   LIN {X -9.322, Y 41.876, Z 87.550} C_DIS
   LIN {X -9.208, Y 43.312, Z 87.550} C_DIS
   LIN {X -9.178, Y 43.420, Z 87.550} C_DIS
   LIN {X -8.370, Y 44.918, Z 87.550} C_DIS
   LIN {X -6.846, Y 45.773, Z 87.550} C_DIS
   LIN {X -6.068, Y 46.221, Z 87.550} C_DIS
   LIN {X -5.087, Y 46.175, Z 87.550} C_DIS
   LIN {X -4.325, Y 46.141, Z 87.550}
   LaserEnd_Ext()
   LIN {X -8.280, Y 42.370, Z 87.550}
   LaserStart_Ext()
   LIN {X -8.280, Y 41.871, Z 87.550}
   LaserEnd_Ext()
   LIN {X -7.280, Y 39.330, Z 87.550}
   LaserStart_Ext()
   LIN {X -7.280, Y 44.383, Z 87.550}
   LaserEnd_Ext()
   LIN {X -6.280, Y 44.945, Z 87.550}
   LaserStart_Ext()
   LIN {X -6.280, Y 36.969, Z 87.550}
   LaserEnd_Ext()
   LIN {X -5.280, Y -20.988, Z 87.550}
   LaserStart_Ext()
   LIN {X -5.280, Y -16.273, Z 87.550}
   LaserEnd_Ext()
   LIN {X -5.280, Y 34.366, Z 87.550}
   LaserStart_Ext()
   LIN {X -5.280, Y 45.183, Z 87.550}
   LaserEnd_Ext()
   LIN {X -4.280, Y 44.988, Z 87.550}
   LaserStart_Ext()
   LIN {X -4.280, Y 31.324, Z 87.550}
   LaserEnd_Ext()
   LIN {X -4.280, Y -13.176, Z 87.550}
   LaserStart_Ext()
   LIN {X -4.280, Y -23.277, Z 87.550}
   LaserEnd_Ext()
   LIN {X -3.280, Y -24.526, Z 87.550}
   LaserStart_Ext()
   LIN {X -3.280, Y -20.919, Z 87.550}
   LaserEnd_Ext()
   LIN {X -3.280, Y -17.023, Z 87.550}
   LaserStart_Ext()
   LIN {X -3.280, Y -9.752, Z 87.550}
   LaserEnd_Ext()
   LIN {X -3.280, Y 27.844, Z 87.550}
   LaserStart_Ext()
   LIN {X -3.280, Y 44.352, Z 87.550}
   LaserEnd_Ext()
   LIN {X -2.280, Y 42.864, Z 87.550}
   LaserStart_Ext()
   LIN {X -2.280, Y 23.421, Z 87.550}
   LaserEnd_Ext()
   LIN {X -2.280, Y -5.420, Z 87.550}
   LaserStart_Ext()
   LIN {X -2.280, Y -15.048, Z 87.550}
   LaserEnd_Ext()
   LIN {X -2.280, Y -22.581, Z 87.550}
   LaserStart_Ext()
   LIN {X -2.280, Y -25.295, Z 87.550}
   LaserEnd_Ext()
   LIN {X -1.280, Y -25.911, Z 87.550}
   LaserStart_Ext()
   LIN {X -1.280, Y -23.637, Z 87.550}
   LaserEnd_Ext()
   LIN {X -1.280, Y -13.980, Z 87.550}
   LaserStart_Ext()
   LIN {X -1.280, Y 1.203, Z 87.550}
   LaserEnd_Ext()
   LIN {X -1.280, Y 16.034, Z 87.550}
   LaserStart_Ext()
   LIN {X -1.280, Y 40.953, Z 87.550}
   LaserEnd_Ext()
   LIN {X -0.280, Y 38.939, Z 87.550}
   LaserStart_Ext()
   LIN {X -0.280, Y -13.537, Z 87.550}
   LaserEnd_Ext()
   LIN {X -0.280, Y -24.134, Z 87.550}
   LaserStart_Ext()
   LIN {X -0.280, Y -26.154, Z 87.550}
   LaserEnd_Ext()
   LIN {X 0.720, Y -26.397, Z 87.550}
   LaserStart_Ext()
   LIN {X 0.720, Y -24.611, Z 87.550}
   LaserEnd_Ext()
   LIN {X 0.720, Y -13.095, Z 87.550}
   LaserStart_Ext()
   LIN {X 0.720, Y 36.811, Z 87.550}
   LaserEnd_Ext()
   LIN {X 1.720, Y 34.552, Z 87.550}
   LaserStart_Ext()
   LIN {X 1.720, Y -12.865, Z 87.550}
   LaserEnd_Ext()
   LIN {X 1.720, Y -24.679, Z 87.550}
   LaserStart_Ext()
   LIN {X 1.720, Y -26.645, Z 87.550}
   LaserEnd_Ext()
   LIN {X 2.720, Y -26.731, Z 87.550}
   LaserStart_Ext()
   LIN {X 2.720, Y -24.716, Z 87.550}
   LaserEnd_Ext()
   LIN {X 2.720, Y -12.903, Z 87.550}
   LaserStart_Ext()
   LIN {X 2.720, Y 32.147, Z 87.550}
   LaserEnd_Ext()
   LIN {X 3.720, Y 29.606, Z 87.550}
   LaserStart_Ext()
   LIN {X 3.720, Y -12.955, Z 87.550}
   LaserEnd_Ext()
   LIN {X 3.720, Y -24.543, Z 87.550}
   LaserStart_Ext()
   LIN {X 3.720, Y -26.549, Z 87.550}
   LaserEnd_Ext()
   LIN {X 4.720, Y -26.367, Z 87.550}
   LaserStart_Ext()
   LIN {X 4.720, Y -24.134, Z 87.550}
   LaserEnd_Ext()
   LIN {X 4.720, Y -13.416, Z 87.550}
   LaserStart_Ext()
   LIN {X 4.720, Y 26.609, Z 87.550}
   LaserEnd_Ext()
   LIN {X 5.720, Y 23.635, Z 87.550}
   LaserStart_Ext()
   LIN {X 5.720, Y -13.918, Z 87.550}
   LaserEnd_Ext()
   LIN {X 5.720, Y -23.685, Z 87.550}
   LaserStart_Ext()
   LIN {X 5.720, Y -25.868, Z 87.550}
   LaserEnd_Ext()
   LIN {X 6.720, Y -25.325, Z 87.550}
   LaserStart_Ext()
   LIN {X 6.720, Y -22.621, Z 87.550}
   LaserEnd_Ext()
   LIN {X 6.720, Y -14.966, Z 87.550}
   LaserStart_Ext()
   LIN {X 6.720, Y 20.268, Z 87.550}
   LaserEnd_Ext()
   LIN {X 7.720, Y 16.143, Z 87.550}
   LaserStart_Ext()
   LIN {X 7.720, Y -16.327, Z 87.550}
   LaserEnd_Ext()
   LIN {X 7.720, Y -21.000, Z 87.550}
   LaserStart_Ext()
   LIN {X 7.720, Y -24.463, Z 87.550}
   LaserEnd_Ext()
   LIN {X 8.720, Y -23.296, Z 87.550}
   LaserStart_Ext()
   LIN {X 8.720, Y 12.020, Z 87.550}
   LaserEnd_Ext()
   LIN {X 9.720, Y 5.409, Z 87.550}
   LaserStart_Ext()
   LIN {X 9.720, Y -21.071, Z 87.550}
   LaserEnd_Ext()
   LIN {X 10.720, Y -10.941, Z 87.550}
   LaserStart_Ext()
   LIN {X 10.720, Y -7.263, Z 87.550}
   LaserEnd_Ext()
   LIN {X -2.101, Y -21.081, Z 88.400}
   LaserStart_Ext()
   LIN {X -2.327, Y -20.250, Z 88.400} C_DIS
   LIN {X -2.653, Y -19.069, Z 88.400} C_DIS
   LIN {X -2.140, Y -16.745, Z 88.400} C_DIS
   LIN {X -2.058, Y -16.383, Z 88.400} C_DIS
   LIN {X -1.960, Y -16.269, Z 88.400} C_DIS
   LIN {X -0.730, Y -14.804, Z 88.400} C_DIS
   LIN {X 1.550, Y -13.800, Z 88.400} C_DIS
   LIN {X 2.406, Y -13.830, Z 88.400} C_DIS
   LIN {X 3.592, Y -13.874, Z 88.400} C_DIS
   LIN {X 4.404, Y -14.282, Z 88.400} C_DIS
   LIN {X 5.494, Y -14.823, Z 88.400} C_DIS
   LIN {X 6.466, Y -16.137, Z 88.400} C_DIS
   LIN {X 7.004, Y -16.869, Z 88.400} C_DIS
   LIN {X 7.127, Y -17.688, Z 88.400} C_DIS
   LIN {X 7.338, Y -19.054, Z 88.400} C_DIS
   LIN {X 6.967, Y -20.266, Z 88.400} C_DIS
   LIN {X 6.671, Y -21.222, Z 88.400} C_DIS
   LIN {X 5.735, Y -22.242, Z 88.400} C_DIS
   LIN {X 5.196, Y -22.834, Z 88.400} C_DIS
   LIN {X 4.756, Y -23.018, Z 88.400} C_DIS
   LIN {X 3.171, Y -23.668, Z 88.400} C_DIS
   LIN {X 1.356, Y -23.607, Z 88.400} C_DIS
   LIN {X 1.086, Y -23.596, Z 88.400} C_DIS
   LIN {X 0.744, Y -23.427, Z 88.400} C_DIS
   LIN {X -0.767, Y -22.681, Z 88.400} C_DIS
   LIN {X -1.591, Y -21.695, Z 88.400} C_DIS
   LIN {X -2.101, Y -21.081, Z 88.400}
   LaserEnd_Ext()
   LIN {X -1.865, Y -26.739, Z 88.400}
   LaserStart_Ext()
   LIN {X -2.207, Y -26.496, Z 88.400} C_DIS
   LIN {X -4.280, Y -24.904, Z 88.400} C_DIS
   LIN {X -5.389, Y -23.237, Z 88.400} C_DIS
   LIN {X -5.889, Y -22.475, Z 88.400} C_DIS
   LIN {X -6.157, Y -21.214, Z 88.400} C_DIS
   LIN {X -6.672, Y -18.848, Z 88.400} C_DIS
   LIN {X -6.289, Y -16.613, Z 88.400} C_DIS
   LIN {X -6.132, Y -15.724, Z 88.400} C_DIS
   LIN {X -5.888, Y -15.002, Z 88.400} C_DIS
   LIN {X -5.036, Y -12.454, Z 88.400} C_DIS
   LIN {X -4.260, Y -9.716, Z 88.400} C_DIS
   LIN {X -4.130, Y -9.256, Z 88.400} C_DIS
   LIN {X -4.052, Y -8.927, Z 88.400} C_DIS
   LIN {X -3.419, Y -6.256, Z 88.400} C_DIS
   LIN {X -3.129, Y -4.745, Z 88.400} C_DIS
   LIN {X -2.837, Y -3.225, Z 88.400} C_DIS
   LIN {X -2.519, Y -1.124, Z 88.400} C_DIS
   LIN {X -2.431, Y -0.548, Z 88.400} C_DIS
   LIN {X -1.994, Y 3.966, Z 88.400} C_DIS
   LIN {X -1.892, Y 5.625, Z 88.400} C_DIS
   LIN {X -1.905, Y 12.231, Z 88.400} C_DIS
   LIN {X -2.343, Y 17.044, Z 88.400} C_DIS
   LIN {X -3.185, Y 22.879, Z 88.400} C_DIS
   LIN {X -4.399, Y 28.248, Z 88.400} C_DIS
   LIN {X -4.637, Y 29.079, Z 88.400} C_DIS
   LIN {X -5.862, Y 32.955, Z 88.400} C_DIS
   LIN {X -5.956, Y 33.234, Z 88.400} C_DIS
   LIN {X -6.386, Y 34.380, Z 88.400} C_DIS
   LIN {X -6.924, Y 35.827, Z 88.400} C_DIS
   LIN {X -7.316, Y 36.776, Z 88.400} C_DIS
   LIN {X -7.831, Y 38.016, Z 88.400} C_DIS
   LIN {X -8.303, Y 39.073, Z 88.400} C_DIS
   LIN {X -8.483, Y 39.477, Z 88.400} C_DIS
   LIN {X -8.577, Y 39.682, Z 88.400} C_DIS
   LIN {X -9.008, Y 40.612, Z 88.400} C_DIS
   LIN {X -9.347, Y 41.838, Z 88.400} C_DIS
   LIN {X -9.397, Y 42.016, Z 88.400} C_DIS
   LIN {X -9.375, Y 42.239, Z 88.400} C_DIS
   LIN {X -9.262, Y 43.429, Z 88.400} C_DIS
   LIN {X -8.453, Y 44.892, Z 88.400} C_DIS
   LIN {X -8.396, Y 44.998, Z 88.400} C_DIS
   LIN {X -8.295, Y 45.059, Z 88.400} C_DIS
   LIN {X -6.140, Y 46.258, Z 88.400} C_DIS
   LIN {X -5.430, Y 46.228, Z 88.400} C_DIS
   LIN {X -4.398, Y 46.181, Z 88.400} C_DIS
   LIN {X -3.166, Y 45.535, Z 88.400} C_DIS
   LIN {X -2.858, Y 45.374, Z 88.400} C_DIS
   LIN {X -2.697, Y 45.180, Z 88.400} C_DIS
   LIN {X -1.925, Y 44.237, Z 88.400} C_DIS
   LIN {X -1.257, Y 43.001, Z 88.400} C_DIS
   LIN {X -1.154, Y 42.804, Z 88.400} C_DIS
   LIN {X -0.334, Y 41.232, Z 88.400} C_DIS
   LIN {X 0.389, Y 39.778, Z 88.400} C_DIS
   LIN {X 0.732, Y 39.087, Z 88.400} C_DIS
   LIN {X 0.977, Y 38.576, Z 88.400} C_DIS
   LIN {X 2.267, Y 35.768, Z 88.400} C_DIS
   LIN {X 2.837, Y 34.460, Z 88.400} C_DIS
   LIN {X 4.233, Y 31.014, Z 88.400} C_DIS
   LIN {X 4.570, Y 30.191, Z 88.400} C_DIS
   LIN {X 4.734, Y 29.722, Z 88.400} C_DIS
   LIN {X 7.364, Y 21.900, Z 88.400} C_DIS
   LIN {X 8.161, Y 18.532, Z 88.400} C_DIS
   LIN {X 9.659, Y 12.653, Z 88.400} C_DIS
   LIN {X 10.596, Y 6.682, Z 88.400} C_DIS
   LIN {X 11.255, Y 1.954, Z 88.400} C_DIS
   LIN {X 11.382, Y -0.482, Z 88.400} C_DIS
   LIN {X 11.492, Y -1.843, Z 88.400} C_DIS
   LIN {X 11.725, Y -4.721, Z 88.400} C_DIS
   LIN {X 11.784, Y -8.079, Z 88.400} C_DIS
   LIN {X 11.812, Y -9.507, Z 88.400} C_DIS
   LIN {X 11.807, Y -9.910, Z 88.400} C_DIS
   LIN {X 11.734, Y -13.310, Z 88.400} C_DIS
   LIN {X 11.644, Y -15.135, Z 88.400} C_DIS
   LIN {X 11.582, Y -16.267, Z 88.400} C_DIS
   LIN {X 11.486, Y -17.425, Z 88.400} C_DIS
   LIN {X 11.326, Y -19.519, Z 88.400} C_DIS
   LIN {X 10.716, Y -21.461, Z 88.400} C_DIS
   LIN {X 10.154, Y -23.186, Z 88.400} C_DIS
   LIN {X 8.060, Y -25.630, Z 88.400} C_DIS
   LIN {X 7.954, Y -25.756, Z 88.400} C_DIS
   LIN {X 7.764, Y -25.857, Z 88.400} C_DIS
   LIN {X 5.067, Y -27.308, Z 88.400} C_DIS
   LIN {X 3.728, Y -27.551, Z 88.400} C_DIS
   LIN {X 1.570, Y -27.601, Z 88.400} C_DIS
   LIN {X -1.865, Y -26.739, Z 88.400}
   LaserEnd_Ext()
   LIN {X 4.690, Y -26.360, Z 88.400}
   LaserStart_Ext()
   LIN {X 0.734, Y -26.360, Z 88.400}
   LaserEnd_Ext()
   LIN {X -2.044, Y -25.360, Z 88.400}
   LaserStart_Ext()
   LIN {X 6.576, Y -25.360, Z 88.400}
   LaserEnd_Ext()
   LIN {X 7.832, Y -24.360, Z 88.400}
   LaserStart_Ext()
   LIN {X 4.118, Y -24.360, Z 88.400}
   LaserEnd_Ext()
   LIN {X 0.375, Y -24.360, Z 88.400}
   LaserStart_Ext()
   LIN {X -3.346, Y -24.360, Z 88.400}
   LaserEnd_Ext()
   LIN {X -4.106, Y -23.360, Z 88.400}
   LaserStart_Ext()
   LIN {X -1.499, Y -23.360, Z 88.400}
   LaserEnd_Ext()
   LIN {X 6.070, Y -23.360, Z 88.400}
   LaserStart_Ext()
   LIN {X 8.688, Y -23.360, Z 88.400}
   LaserEnd_Ext()
   LIN {X 9.371, Y -22.360, Z 88.400}
   LaserStart_Ext()
   LIN {X 6.984, Y -22.360, Z 88.400}
   LaserEnd_Ext()
   LIN {X -2.339, Y -22.360, Z 88.400}
   LaserStart_Ext()
   LIN {X -4.768, Y -22.360, Z 88.400}
   LaserEnd_Ext()
   LIN {X -5.103, Y -21.360, Z 88.400}
   LaserStart_Ext()
   LIN {X -3.060, Y -21.360, Z 88.400}
   LaserEnd_Ext()
   LIN {X 7.675, Y -21.360, Z 88.400}
   LaserStart_Ext()
   LIN {X 9.697, Y -21.360, Z 88.400}
   LaserEnd_Ext()
   LIN {X 10.014, Y -20.360, Z 88.400}
   LaserStart_Ext()
   LIN {X 7.984, Y -20.360, Z 88.400}
   LaserEnd_Ext()
   LIN {X -3.334, Y -20.360, Z 88.400}
   LaserStart_Ext()
   LIN {X -5.319, Y -20.360, Z 88.400}
   LaserEnd_Ext()
   LIN {X -5.537, Y -19.360, Z 88.400}
   LaserStart_Ext()
   LIN {X -3.610, Y -19.360, Z 88.400}
   LaserEnd_Ext()
   LIN {X 8.290, Y -19.360, Z 88.400}
   LaserStart_Ext()
   LIN {X 10.328, Y -19.360, Z 88.400}
   LaserEnd_Ext()
   LIN {X 10.412, Y -18.360, Z 88.400}
   LaserStart_Ext()
   LIN {X 8.243, Y -18.360, Z 88.400}
   LaserEnd_Ext()
   LIN {X -3.521, Y -18.360, Z 88.400}
   LaserStart_Ext()
   LIN {X -5.574, Y -18.360, Z 88.400}
   LaserEnd_Ext()
   LIN {X -5.402, Y -17.360, Z 88.400}
   LaserStart_Ext()
   LIN {X -3.300, Y -17.360, Z 88.400}
   LaserEnd_Ext()
   LIN {X 8.089, Y -17.360, Z 88.400}
   LaserStart_Ext()
   LIN {X 10.488, Y -17.360, Z 88.400}
   LaserEnd_Ext()
   LIN {X 10.571, Y -16.360, Z 88.400}
   LaserStart_Ext()
   LIN {X 7.864, Y -16.360, Z 88.400}
   LaserEnd_Ext()
   LIN {X -3.078, Y -16.360, Z 88.400}
   LaserStart_Ext()
   LIN {X -5.228, Y -16.360, Z 88.400}
   LaserEnd_Ext()
   LIN {X -4.953, Y -15.360, Z 88.400}
   LaserStart_Ext()
   LIN {X -2.503, Y -15.360, Z 88.400}
   LaserEnd_Ext()
   LIN {X 7.135, Y -15.360, Z 88.400}
   LaserStart_Ext()
   LIN {X 10.630, Y -15.360, Z 88.400}
   LaserEnd_Ext()
   LIN {X 10.681, Y -14.360, Z 88.400}
   LaserStart_Ext()
   LIN {X 6.395, Y -14.360, Z 88.400}
   LaserEnd_Ext()
   LIN {X -1.663, Y -14.360, Z 88.400}
   LaserStart_Ext()
   LIN {X -4.619, Y -14.360, Z 88.400}
   LaserEnd_Ext()
   LIN {X -4.284, Y -13.360, Z 88.400}
   LaserStart_Ext()
   LIN {X 0.068, Y -13.360, Z 88.400}
   LaserEnd_Ext()
   LIN {X 4.797, Y -13.360, Z 88.400}
   LaserStart_Ext()
   LIN {X 10.730, Y -13.360, Z 88.400}
   LaserEnd_Ext()
   LIN {X 10.754, Y -12.360, Z 88.400}
   LaserStart_Ext()
   LIN {X -3.970, Y -12.360, Z 88.400}
   LaserEnd_Ext()
   LIN {X -3.687, Y -11.360, Z 88.400}
   LaserStart_Ext()
   LIN {X 10.775, Y -11.360, Z 88.400}
   LaserEnd_Ext()
   LIN {X 10.797, Y -10.360, Z 88.400}
   LaserStart_Ext()
   LIN {X -3.403, Y -10.360, Z 88.400}
   LaserEnd_Ext()
   LIN {X -3.127, Y -9.360, Z 88.400}
   LaserStart_Ext()
   LIN {X 10.809, Y -9.360, Z 88.400}
   LaserEnd_Ext()
   LIN {X 10.789, Y -8.360, Z 88.400}
   LaserStart_Ext()
   LIN {X -2.890, Y -8.360, Z 88.400}
   LaserEnd_Ext()
   LIN {X -2.653, Y -7.360, Z 88.400}
   LaserStart_Ext()
   LIN {X 10.771, Y -7.360, Z 88.400}
   LaserEnd_Ext()
   LIN {X 10.754, Y -6.360, Z 88.400}
   LaserStart_Ext()
   LIN {X -2.421, Y -6.360, Z 88.400}
   LaserEnd_Ext()
   LIN {X -2.229, Y -5.360, Z 88.400}
   LaserStart_Ext()
   LIN {X 10.736, Y -5.360, Z 88.400}
   LaserEnd_Ext()
   LIN {X 10.693, Y -4.360, Z 88.400}
   LaserStart_Ext()
   LIN {X -2.037, Y -4.360, Z 88.400}
   LaserEnd_Ext()
   LIN {X -1.846, Y -3.360, Z 88.400}
   LaserStart_Ext()
   LIN {X 10.612, Y -3.360, Z 88.400}
   LaserEnd_Ext()
   LIN {X 10.531, Y -2.360, Z 88.400}
   LaserStart_Ext()
   LIN {X -1.694, Y -2.360, Z 88.400}
   LaserEnd_Ext()
   LIN {X -1.543, Y -1.360, Z 88.400}
   LaserStart_Ext()
   LIN {X 10.450, Y -1.360, Z 88.400}
   LaserEnd_Ext()
   LIN {X 10.375, Y -0.360, Z 88.400}
   LaserStart_Ext()
   LIN {X -1.408, Y -0.360, Z 88.400}
   LaserEnd_Ext()
   LIN {X -1.311, Y 0.640, Z 88.400}
   LaserStart_Ext()
   LIN {X 10.322, Y 0.640, Z 88.400}
   LaserEnd_Ext()
   LIN {X 10.270, Y 1.640, Z 88.400}
   LaserStart_Ext()
   LIN {X -1.214, Y 1.640, Z 88.400}
   LaserEnd_Ext()
   LIN {X -1.118, Y 2.640, Z 88.400}
   LaserStart_Ext()
   LIN {X 10.149, Y 2.640, Z 88.400}
   LaserEnd_Ext()
   LIN {X 10.010, Y 3.640, Z 88.400}
   LaserStart_Ext()
   LIN {X -1.021, Y 3.640, Z 88.400}
   LaserEnd_Ext()
   LIN {X -0.951, Y 4.640, Z 88.400}
   LaserStart_Ext()
   LIN {X 9.871, Y 4.640, Z 88.400}
   LaserEnd_Ext()
   LIN {X 9.732, Y 5.640, Z 88.400}
   LaserStart_Ext()
   LIN {X -0.892, Y 5.640, Z 88.400}
   LaserEnd_Ext()
   LIN {X -0.894, Y 6.640, Z 88.400}
   LaserStart_Ext()
   LIN {X 9.591, Y 6.640, Z 88.400}
   LaserEnd_Ext()
   LIN {X 9.434, Y 7.640, Z 88.400}
   LaserStart_Ext()
   LIN {X -0.896, Y 7.640, Z 88.400}
   LaserEnd_Ext()
   LIN {X -0.898, Y 8.640, Z 88.400}
   LaserStart_Ext()
   LIN {X 9.277, Y 8.640, Z 88.400}
   LaserEnd_Ext()
   LIN {X 9.120, Y 9.640, Z 88.400}
   LaserStart_Ext()
   LIN {X -0.900, Y 9.640, Z 88.400}
   LaserEnd_Ext()
   LIN {X -0.902, Y 10.640, Z 88.400}
   LaserStart_Ext()
   LIN {X 8.963, Y 10.640, Z 88.400}
   LaserEnd_Ext()
   LIN {X 8.806, Y 11.640, Z 88.400}
   LaserStart_Ext()
   LIN {X -0.904, Y 11.640, Z 88.400}
   LaserEnd_Ext()
   LIN {X -0.938, Y 12.640, Z 88.400}
   LaserStart_Ext()
   LIN {X 8.630, Y 12.640, Z 88.400}
   LaserEnd_Ext()
   LIN {X 8.376, Y 13.640, Z 88.400}
   LaserStart_Ext()
   LIN {X -1.029, Y 13.640, Z 88.400}
   LaserEnd_Ext()
   LIN {X -1.120, Y 14.640, Z 88.400}
   LaserStart_Ext()
   LIN {X 8.121, Y 14.640, Z 88.400}
   LaserEnd_Ext()
   LIN {X 7.866, Y 15.640, Z 88.400}
   LaserStart_Ext()
   LIN {X -1.211, Y 15.640, Z 88.400}
   LaserEnd_Ext()
   LIN {X -1.302, Y 16.640, Z 88.400}
   LaserStart_Ext()
   LIN {X 7.611, Y 16.640, Z 88.400}
   LaserEnd_Ext()
   LIN {X 7.356, Y 17.640, Z 88.400}
   LaserStart_Ext()
   LIN {X -1.419, Y 17.640, Z 88.400}
   LaserEnd_Ext()
   LIN {X -1.563, Y 18.640, Z 88.400}
   LaserStart_Ext()
   LIN {X 7.108, Y 18.640, Z 88.400}
   LaserEnd_Ext()
   LIN {X 6.871, Y 19.640, Z 88.400}
   LaserStart_Ext()
   LIN {X -1.707, Y 19.640, Z 88.400}
   LaserEnd_Ext()
   LIN {X -1.852, Y 20.640, Z 88.400}
   LaserStart_Ext()
   LIN {X 6.635, Y 20.640, Z 88.400}
   LaserEnd_Ext()
   LIN {X 6.397, Y 21.640, Z 88.400}
   LaserStart_Ext()
   LIN {X -1.996, Y 21.640, Z 88.400}
   LaserEnd_Ext()
   LIN {X -2.141, Y 22.640, Z 88.400}
   LaserStart_Ext()
   LIN {X 6.060, Y 22.640, Z 88.400}
   LaserEnd_Ext()
   LIN {X 5.724, Y 23.640, Z 88.400}
   LaserStart_Ext()
   LIN {X -2.332, Y 23.640, Z 88.400}
   LaserEnd_Ext()
   LIN {X -2.558, Y 24.640, Z 88.400}
   LaserStart_Ext()
   LIN {X 5.388, Y 24.640, Z 88.400}
   LaserEnd_Ext()
   LIN {X 5.052, Y 25.640, Z 88.400}
   LaserStart_Ext()
   LIN {X -2.784, Y 25.640, Z 88.400}
   LaserEnd_Ext()
   LIN {X -3.010, Y 26.640, Z 88.400}
   LaserStart_Ext()
   LIN {X 4.715, Y 26.640, Z 88.400}
   LaserEnd_Ext()
   LIN {X 4.379, Y 27.640, Z 88.400}
   LaserStart_Ext()
   LIN {X -3.237, Y 27.640, Z 88.400}
   LaserEnd_Ext()
   LIN {X -3.471, Y 28.640, Z 88.400}
   LaserStart_Ext()
   LIN {X 4.043, Y 28.640, Z 88.400}
   LaserEnd_Ext()
   LIN {X 3.703, Y 29.640, Z 88.400}
   LaserStart_Ext()
   LIN {X -3.766, Y 29.640, Z 88.400}
   LaserEnd_Ext()
   LIN {X -4.082, Y 30.640, Z 88.400}
   LaserStart_Ext()
   LIN {X 3.306, Y 30.640, Z 88.400}
   LaserEnd_Ext()
   LIN {X 2.900, Y 31.640, Z 88.400}
   LaserStart_Ext()
   LIN {X -4.398, Y 31.640, Z 88.400}
   LaserEnd_Ext()
   LIN {X -4.714, Y 32.640, Z 88.400}
   LaserStart_Ext()
   LIN {X 2.495, Y 32.640, Z 88.400}
   LaserEnd_Ext()
   LIN {X 2.090, Y 33.640, Z 88.400}
   LaserStart_Ext()
   LIN {X -5.040, Y 33.640, Z 88.400}
   LaserEnd_Ext()
   LIN {X -5.415, Y 34.640, Z 88.400}
   LaserStart_Ext()
   LIN {X 1.668, Y 34.640, Z 88.400}
   LaserEnd_Ext()
   LIN {X 1.226, Y 35.640, Z 88.400}
   LaserStart_Ext()
   LIN {X -5.788, Y 35.640, Z 88.400}
   LaserEnd_Ext()
   LIN {X -6.178, Y 36.640, Z 88.400}
   LaserStart_Ext()
   LIN {X 0.766, Y 36.640, Z 88.400}
   LaserEnd_Ext()
   LIN {X 0.306, Y 37.640, Z 88.400}
   LaserStart_Ext()
   LIN {X -6.592, Y 37.640, Z 88.400}
   LaserEnd_Ext()
   LIN {X -7.014, Y 38.640, Z 88.400}
   LaserStart_Ext()
   LIN {X -0.163, Y 38.640, Z 88.400}
   LaserEnd_Ext()
   LIN {X -0.659, Y 39.640, Z 88.400}
   LaserStart_Ext()
   LIN {X -7.461, Y 39.640, Z 88.400}
   LaserEnd_Ext()
   LIN {X -7.919, Y 40.640, Z 88.400}
   LaserStart_Ext()
   LIN {X -1.156, Y 40.640, Z 88.400}
   LaserEnd_Ext()
   LIN {X -1.674, Y 41.640, Z 88.400}
   LaserStart_Ext()
   LIN {X -8.255, Y 41.640, Z 88.400}
   LaserEnd_Ext()
   LIN {X -8.333, Y 42.640, Z 88.400}
   LaserStart_Ext()
   LIN {X -2.199, Y 42.640, Z 88.400}
   LaserEnd_Ext()
   LIN {X -2.739, Y 43.640, Z 88.400}
   LaserStart_Ext()
   LIN {X -8.003, Y 43.640, Z 88.400}
   LaserEnd_Ext()
   LIN {X -6.992, Y 44.640, Z 88.400}
   LaserStart_Ext()
   LIN {X -3.612, Y 44.640, Z 88.400}
   LaserEnd_Ext()
   LIN {X -1.592, Y -21.537, Z 89.250}
   LaserStart_Ext()
   LIN {X -2.015, Y -21.035, Z 89.250} C_DIS
   LIN {X -2.194, Y -20.394, Z 89.250} C_DIS
   LIN {X -2.572, Y -19.024, Z 89.250} C_DIS
   LIN {X -2.278, Y -17.692, Z 89.250} C_DIS
   LIN {X -1.967, Y -16.308, Z 89.250} C_DIS
   LIN {X -0.892, Y -15.038, Z 89.250} C_DIS
   LIN {X -0.644, Y -14.743, Z 89.250} C_DIS
   LIN {X 1.620, Y -13.745, Z 89.250} C_DIS
   LIN {X 3.253, Y -13.802, Z 89.250} C_DIS
   LIN {X 3.661, Y -13.815, Z 89.250} C_DIS
   LIN {X 4.151, Y -14.057, Z 89.250} C_DIS
   LIN {X 5.565, Y -14.759, Z 89.250} C_DIS
   LIN {X 6.551, Y -16.091, Z 89.250} C_DIS
   LIN {X 7.080, Y -16.801, Z 89.250} C_DIS
   LIN {X 7.186, Y -17.471, Z 89.250} C_DIS
   LIN {X 7.420, Y -18.985, Z 89.250} C_DIS
   LIN {X 6.909, Y -20.653, Z 89.250} C_DIS
   LIN {X 6.757, Y -21.155, Z 89.250} C_DIS
   LIN {X 6.481, Y -21.460, Z 89.250} C_DIS
   LIN {X 5.289, Y -22.769, Z 89.250} C_DIS
   LIN {X 3.705, Y -23.429, Z 89.250} C_DIS
   LIN {X 3.268, Y -23.608, Z 89.250} C_DIS
   LIN {X 2.586, Y -23.585, Z 89.250} C_DIS
   LIN {X 1.178, Y -23.542, Z 89.250} C_DIS
   LIN {X 0.300, Y -23.114, Z 89.250} C_DIS
   LIN {X -0.677, Y -22.631, Z 89.250} C_DIS
   LIN {X -1.592, Y -21.537, Z 89.250}
   LaserEnd_Ext()
   LIN {X -5.998, Y 33.271, Z 89.250}
   LaserStart_Ext()
   LIN {X -5.632, Y 32.183, Z 89.250} C_DIS
   LIN {X -4.767, Y 29.446, Z 89.250} C_DIS
   LIN {X -4.321, Y 27.887, Z 89.250} C_DIS
   LIN {X -3.278, Y 23.278, Z 89.250} C_DIS
   LIN {X -2.195, Y 15.771, Z 89.250} C_DIS
   LIN {X -1.905, Y 12.581, Z 89.250} C_DIS
   LIN {X -1.889, Y 5.163, Z 89.250} C_DIS
   LIN {X -1.949, Y 4.193, Z 89.250} C_DIS
   LIN {X -2.359, Y -0.048, Z 89.250} C_DIS
   LIN {X -2.418, Y -0.675, Z 89.250} C_DIS
   LIN {X -2.505, Y -1.257, Z 89.250} C_DIS
   LIN {X -2.823, Y -3.356, Z 89.250} C_DIS
   LIN {X -2.949, Y -4.013, Z 89.250} C_DIS
   LIN {X -3.404, Y -6.387, Z 89.250} C_DIS
   LIN {X -3.835, Y -8.202, Z 89.250} C_DIS
   LIN {X -4.113, Y -9.379, Z 89.250} C_DIS
   LIN {X -4.579, Y -11.021, Z 89.250} C_DIS
   LIN {X -5.020, Y -12.577, Z 89.250} C_DIS
   LIN {X -5.817, Y -14.962, Z 89.250} C_DIS
   LIN {X -6.058, Y -15.688, Z 89.250} C_DIS
   LIN {X -6.170, Y -16.361, Z 89.250} C_DIS
   LIN {X -6.591, Y -18.813, Z 89.250} C_DIS
   LIN {X -5.908, Y -21.949, Z 89.250} C_DIS
   LIN {X -5.799, Y -22.438, Z 89.250} C_DIS
   LIN {X -5.547, Y -22.814, Z 89.250} C_DIS
   LIN {X -4.184, Y -24.863, Z 89.250} C_DIS
   LIN {X -2.991, Y -25.779, Z 89.250} C_DIS
   LIN {X -1.597, Y -26.769, Z 89.250} C_DIS
   LIN {X 1.038, Y -27.430, Z 89.250} C_DIS
   LIN {X 4.803, Y -27.343, Z 89.250} C_DIS
   LIN {X 4.970, Y -27.313, Z 89.250} C_DIS
   LIN {X 5.307, Y -27.132, Z 89.250} C_DIS
   LIN {X 7.191, Y -26.181, Z 89.250} C_DIS
   LIN {X 8.065, Y -25.674, Z 89.250} C_DIS
   LIN {X 9.619, Y -23.837, Z 89.250} C_DIS
   LIN {X 10.254, Y -23.096, Z 89.250} C_DIS
   LIN {X 10.425, Y -22.572, Z 89.250} C_DIS
   LIN {X 11.409, Y -19.441, Z 89.250} C_DIS
   LIN {X 11.649, Y -16.305, Z 89.250} C_DIS
   LIN {X 11.657, Y -16.188, Z 89.250} C_DIS
   LIN {X 11.665, Y -16.024, Z 89.250} C_DIS
   LIN {X 11.802, Y -13.231, Z 89.250} C_DIS
   LIN {X 11.847, Y -11.119, Z 89.250} C_DIS
   LIN {X 11.872, Y -9.427, Z 89.250} C_DIS
   LIN {X 11.785, Y -5.074, Z 89.250} C_DIS
   LIN {X 11.773, Y -4.642, Z 89.250} C_DIS
   LIN {X 11.733, Y -4.149, Z 89.250} C_DIS
   LIN {X 11.468, Y -0.870, Z 89.250} C_DIS
   LIN {X 11.383, Y 0.176, Z 89.250} C_DIS
   LIN {X 11.285, Y 2.048, Z 89.250} C_DIS
   LIN {X 10.779, Y 5.683, Z 89.250} C_DIS
   LIN {X 9.699, Y 12.567, Z 89.250} C_DIS
   LIN {X 7.971, Y 19.344, Z 89.250} C_DIS
   LIN {X 7.360, Y 21.930, Z 89.250} C_DIS
   LIN {X 5.341, Y 27.934, Z 89.250} C_DIS
   LIN {X 4.513, Y 30.308, Z 89.250} C_DIS
   LIN {X 2.805, Y 34.476, Z 89.250} C_DIS
   LIN {X 2.660, Y 34.835, Z 89.250} C_DIS
   LIN {X 2.600, Y 34.972, Z 89.250} C_DIS
   LIN {X 2.284, Y 35.660, Z 89.250} C_DIS
   LIN {X 0.845, Y 38.792, Z 89.250} C_DIS
   LIN {X 0.072, Y 40.342, Z 89.250} C_DIS
   LIN {X -0.395, Y 41.282, Z 89.250} C_DIS
   LIN {X -0.599, Y 41.673, Z 89.250} C_DIS
   LIN {X -1.285, Y 42.979, Z 89.250} C_DIS
   LIN {X -1.937, Y 44.181, Z 89.250} C_DIS
   LIN {X -1.992, Y 44.283, Z 89.250} C_DIS
   LIN {X -2.078, Y 44.387, Z 89.250} C_DIS
   LIN {X -2.928, Y 45.418, Z 89.250} C_DIS
   LIN {X -4.144, Y 46.053, Z 89.250} C_DIS
   LIN {X -4.470, Y 46.221, Z 89.250} C_DIS
   LIN {X -5.183, Y 46.251, Z 89.250} C_DIS
   LIN {X -6.213, Y 46.294, Z 89.250} C_DIS
   LIN {X -6.786, Y 45.975, Z 89.250} C_DIS
   LIN {X -8.564, Y 44.907, Z 89.250} C_DIS
   LIN {X -9.211, Y 43.703, Z 89.250} C_DIS
   LIN {X -9.330, Y 43.445, Z 89.250} C_DIS
   LIN {X -9.352, Y 43.152, Z 89.250} C_DIS
   LIN {X -9.459, Y 42.045, Z 89.250} C_DIS
   LIN {X -9.087, Y 40.713, Z 89.250} C_DIS
   LIN {X -9.048, Y 40.601, Z 89.250} C_DIS
   LIN {X -8.539, Y 39.508, Z 89.250} C_DIS
   LIN {X -8.096, Y 38.522, Z 89.250} C_DIS
   LIN {X -7.884, Y 38.049, Z 89.250} C_DIS
   LIN {X -7.522, Y 37.175, Z 89.250} C_DIS
   LIN {X -6.972, Y 35.861, Z 89.250} C_DIS
   LIN {X -6.433, Y 34.432, Z 89.250} C_DIS
   LIN {X -5.998, Y 33.271, Z 89.250}
   LaserEnd_Ext()
   LIN {X 10.602, Y -2.568, Z 89.250}
   LaserStart_Ext()
   LIN {X 10.602, Y -16.881, Z 89.250}
   LaserEnd_Ext()
   LIN {X 9.602, Y -21.855, Z 89.250}
   LaserStart_Ext()
   LIN {X 9.602, Y 6.733, Z 89.250}
   LaserEnd_Ext()
   LIN {X 8.602, Y 12.821, Z 89.250}
   LaserStart_Ext()
   LIN {X 8.602, Y -23.491, Z 89.250}
   LaserEnd_Ext()
   LIN {X 7.602, Y -24.674, Z 89.250}
   LaserStart_Ext()
   LIN {X 7.602, Y -21.687, Z 89.250}
   LaserEnd_Ext()
   LIN {X 7.602, Y -15.828, Z 89.250}
   LaserStart_Ext()
   LIN {X 7.602, Y 16.744, Z 89.250}
   LaserEnd_Ext()
   LIN {X 6.602, Y 20.790, Z 89.250}
   LaserStart_Ext()
   LIN {X 6.602, Y -14.479, Z 89.250}
   LaserEnd_Ext()
   LIN {X 6.602, Y -22.812, Z 89.250}
   LaserStart_Ext()
   LIN {X 6.602, Y -25.358, Z 89.250}
   LaserEnd_Ext()
   LIN {X 5.602, Y -25.863, Z 89.250}
   LaserStart_Ext()
   LIN {X 5.602, Y -23.722, Z 89.250}
   LaserEnd_Ext()
   LIN {X 5.602, Y -13.661, Z 89.250}
   LaserStart_Ext()
   LIN {X 5.602, Y 24.020, Z 89.250}
   LaserEnd_Ext()
   LIN {X 4.602, Y 26.993, Z 89.250}
   LaserStart_Ext()
   LIN {X 4.602, Y -13.164, Z 89.250}
   LaserEnd_Ext()
   LIN {X 4.602, Y -24.138, Z 89.250}
   LaserStart_Ext()
   LIN {X 4.602, Y -26.348, Z 89.250}
   LaserEnd_Ext()
   LIN {X 3.602, Y -26.371, Z 89.250}
   LaserStart_Ext()
   LIN {X 3.602, Y -24.549, Z 89.250}
   LaserEnd_Ext()
   LIN {X 3.602, Y -12.812, Z 89.250}
   LaserStart_Ext()
   LIN {X 3.602, Y 29.884, Z 89.250}
   LaserEnd_Ext()
   LIN {X 2.602, Y 32.335, Z 89.250}
   LaserStart_Ext()
   LIN {X 2.602, Y -12.779, Z 89.250}
   LaserEnd_Ext()
   LIN {X 2.602, Y -24.586, Z 89.250}
   LaserStart_Ext()
   LIN {X 2.602, Y -26.394, Z 89.250}
   LaserEnd_Ext()
   LIN {X 1.602, Y -26.417, Z 89.250}
   LaserStart_Ext()
   LIN {X 1.602, Y -24.556, Z 89.250}
   LaserEnd_Ext()
   LIN {X 1.602, Y -12.746, Z 89.250}
   LaserStart_Ext()
   LIN {X 1.602, Y 34.749, Z 89.250}
   LaserEnd_Ext()
   LIN {X 0.602, Y 36.926, Z 89.250}
   LaserStart_Ext()
   LIN {X 0.602, Y -13.101, Z 89.250}
   LaserEnd_Ext()
   LIN {X 0.602, Y -24.374, Z 89.250}
   LaserStart_Ext()
   LIN {X 0.602, Y -26.289, Z 89.250}
   LaserEnd_Ext()
   LIN {X -0.398, Y -26.039, Z 89.250}
   LaserStart_Ext()
   LIN {X -0.398, Y -23.884, Z 89.250}
   LaserEnd_Ext()
   LIN {X -0.398, Y -13.542, Z 89.250}
   LaserStart_Ext()
   LIN {X -0.398, Y 39.045, Z 89.250}
   LaserEnd_Ext()
   LIN {X -1.398, Y 41.044, Z 89.250}
   LaserStart_Ext()
   LIN {X -1.398, Y 17.252, Z 89.250}
   LaserEnd_Ext()
   LIN {X -1.398, Y -0.512, Z 89.250}
   LaserStart_Ext()
   LIN {X -1.398, Y -14.087, Z 89.250}
   LaserEnd_Ext()
   LIN {X -1.398, Y -23.323, Z 89.250}
   LaserStart_Ext()
   LIN {X -1.398, Y -25.684, Z 89.250}
   LaserEnd_Ext()
   LIN {X -2.398, Y -24.974, Z 89.250}
   LaserStart_Ext()
   LIN {X -2.398, Y -22.133, Z 89.250}
   LaserEnd_Ext()
   LIN {X -2.398, Y -15.270, Z 89.250}
   LaserStart_Ext()
   LIN {X -2.398, Y -6.448, Z 89.250}
   LaserEnd_Ext()
   LIN {X -2.398, Y 23.919, Z 89.250}
   LaserStart_Ext()
   LIN {X -2.398, Y 42.934, Z 89.250}
   LaserEnd_Ext()
   LIN {X -3.398, Y 44.416, Z 89.250}
   LaserStart_Ext()
   LIN {X -3.398, Y 28.299, Z 89.250}
   LaserEnd_Ext()
   LIN {X -3.398, Y -10.523, Z 89.250}
   LaserStart_Ext()
   LIN {X -3.398, Y -18.128, Z 89.250}
   LaserEnd_Ext()
   LIN {X -3.398, Y -19.788, Z 89.250}
   LaserStart_Ext()
   LIN {X -3.398, Y -24.206, Z 89.250}
   LaserEnd_Ext()
   LIN {X -4.398, Y -22.736, Z 89.250}
   LaserStart_Ext()
   LIN {X -4.398, Y -13.871, Z 89.250}
   LaserEnd_Ext()
   LIN {X -4.398, Y 31.598, Z 89.250}
   LaserStart_Ext()
   LIN {X -4.398, Y 45.057, Z 89.250}
   LaserEnd_Ext()
   LIN {X -5.398, Y 45.259, Z 89.250}
   LaserStart_Ext()
   LIN {X -5.398, Y 34.519, Z 89.250}
   LaserEnd_Ext()
   LIN {X -5.398, Y -17.776, Z 89.250}
   LaserStart_Ext()
   LIN {X -5.398, Y -19.590, Z 89.250}
   LaserEnd_Ext()
   LIN {X -6.398, Y 37.080, Z 89.250}
   LaserStart_Ext()
   LIN {X -6.398, Y 45.042, Z 89.250}
   LaserEnd_Ext()
   LIN {X -7.398, Y 44.441, Z 89.250}
   LaserStart_Ext()
   LIN {X -7.398, Y 39.409, Z 89.250}
   LaserEnd_Ext()
   LIN {X -8.398, Y 41.962, Z 89.250}
   LaserStart_Ext()
   LIN {X -8.398, Y 42.631, Z 89.250}
   LaserEnd_Ext()
   LIN {X -0.588, Y -22.582, Z 90.100}
   LaserStart_Ext()
   LIN {X -0.706, Y -22.442, Z 90.100} C_DIS
   LIN {X -1.929, Y -20.988, Z 90.100} C_DIS
   LIN {X -2.435, Y -19.175, Z 90.100} C_DIS
   LIN {X -2.490, Y -18.979, Z 90.100} C_DIS
   LIN {X -2.411, Y -18.632, Z 90.100} C_DIS
   LIN {X -1.870, Y -16.222, Z 90.100} C_DIS
   LIN {X -1.137, Y -15.356, Z 90.100} C_DIS
   LIN {X -0.541, Y -14.668, Z 90.100} C_DIS
   LIN {X 1.101, Y -13.949, Z 90.100} C_DIS
   LIN {X 1.689, Y -13.690, Z 90.100} C_DIS
   LIN {X 2.048, Y -13.702, Z 90.100} C_DIS
   LIN {X 3.731, Y -13.755, Z 90.100} C_DIS
   LIN {X 5.545, Y -14.650, Z 90.100} C_DIS
   LIN {X 5.637, Y -14.695, Z 90.100} C_DIS
   LIN {X 5.712, Y -14.795, Z 90.100} C_DIS
   LIN {X 7.157, Y -16.733, Z 90.100} C_DIS
   LIN {X 7.477, Y -18.758, Z 90.100} C_DIS
   LIN {X 7.501, Y -18.916, Z 90.100} C_DIS
   LIN {X 7.448, Y -19.090, Z 90.100} C_DIS
   LIN {X 6.839, Y -21.095, Z 90.100} C_DIS
   LIN {X 5.739, Y -22.311, Z 90.100} C_DIS
   LIN {X 5.381, Y -22.704, Z 90.100} C_DIS
   LIN {X 4.557, Y -23.047, Z 90.100} C_DIS
   LIN {X 3.363, Y -23.549, Z 90.100} C_DIS
   LIN {X 2.587, Y -23.528, Z 90.100} C_DIS
   LIN {X 1.270, Y -23.488, Z 90.100} C_DIS
   LIN {X -0.388, Y -22.678, Z 90.100} C_DIS
   LIN {X -0.588, Y -22.582, Z 90.100}
   LaserEnd_Ext()
   LIN {X 5.947, Y 26.147, Z 90.100}
   LaserStart_Ext()
   LIN {X 4.456, Y 30.426, Z 90.100} C_DIS
   LIN {X 2.760, Y 34.563, Z 90.100} C_DIS
   LIN {X 2.404, Y 35.337, Z 90.100} C_DIS
   LIN {X 2.319, Y 35.520, Z 90.100} C_DIS
   LIN {X 2.137, Y 35.913, Z 90.100} C_DIS
   LIN {X 0.791, Y 38.845, Z 90.100} C_DIS
   LIN {X 0.241, Y 39.946, Z 90.100} C_DIS
   LIN {X -0.455, Y 41.332, Z 90.100} C_DIS
   LIN {X -1.225, Y 42.790, Z 90.100} C_DIS
   LIN {X -1.349, Y 43.027, Z 90.100} C_DIS
   LIN {X -1.417, Y 43.152, Z 90.100} C_DIS
   LIN {X -2.059, Y 44.329, Z 90.100} C_DIS
   LIN {X -2.945, Y 45.398, Z 90.100} C_DIS
   LIN {X -3.137, Y 45.533, Z 90.100} C_DIS
   LIN {X -4.542, Y 46.261, Z 90.100} C_DIS
   LIN {X -5.406, Y 46.297, Z 90.100} C_DIS
   LIN {X -6.285, Y 46.330, Z 90.100} C_DIS
   LIN {X -8.269, Y 45.094, Z 90.100} C_DIS
   LIN {X -8.733, Y 44.816, Z 90.100} C_DIS
   LIN {X -8.819, Y 44.655, Z 90.100} C_DIS
   LIN {X -9.432, Y 43.321, Z 90.100} C_DIS
   LIN {X -9.512, Y 42.273, Z 90.100} C_DIS
   LIN {X -9.519, Y 42.051, Z 90.100} C_DIS
   LIN {X -9.451, Y 41.825, Z 90.100} C_DIS
   LIN {X -9.126, Y 40.671, Z 90.100} C_DIS
   LIN {X -8.666, Y 39.690, Z 90.100} C_DIS
   LIN {X -8.596, Y 39.538, Z 90.100} C_DIS
   LIN {X -8.461, Y 39.239, Z 90.100} C_DIS
   LIN {X -7.937, Y 38.081, Z 90.100} C_DIS
   LIN {X -7.273, Y 36.500, Z 90.100} C_DIS
   LIN {X -7.020, Y 35.895, Z 90.100} C_DIS
   LIN {X -6.721, Y 35.101, Z 90.100} C_DIS
   LIN {X -6.041, Y 33.311, Z 90.100} C_DIS
   LIN {X -5.401, Y 31.410, Z 90.100} C_DIS
   LIN {X -4.896, Y 29.812, Z 90.100} C_DIS
   LIN {X -4.242, Y 27.527, Z 90.100} C_DIS
   LIN {X -3.371, Y 23.677, Z 90.100} C_DIS
   LIN {X -2.046, Y 14.497, Z 90.100} C_DIS
   LIN {X -1.904, Y 12.930, Z 90.100} C_DIS
   LIN {X -1.886, Y 4.701, Z 90.100} C_DIS
   LIN {X -1.904, Y 4.420, Z 90.100} C_DIS
   LIN {X -2.022, Y 3.193, Z 90.100} C_DIS
   LIN {X -2.377, Y -0.611, Z 90.100} C_DIS
   LIN {X -2.406, Y -0.844, Z 90.100} C_DIS
   LIN {X -2.783, Y -3.326, Z 90.100} C_DIS
   LIN {X -2.808, Y -3.487, Z 90.100} C_DIS
   LIN {X -2.910, Y -4.018, Z 90.100} C_DIS
   LIN {X -3.390, Y -6.517, Z 90.100} C_DIS
   LIN {X -3.617, Y -7.478, Z 90.100} C_DIS
   LIN {X -4.096, Y -9.502, Z 90.100} C_DIS
   LIN {X -4.898, Y -12.326, Z 90.100} C_DIS
   LIN {X -5.004, Y -12.700, Z 90.100} C_DIS
   LIN {X -5.195, Y -13.272, Z 90.100} C_DIS
   LIN {X -5.984, Y -15.651, Z 90.100} C_DIS
   LIN {X -6.352, Y -17.858, Z 90.100} C_DIS
   LIN {X -6.509, Y -18.778, Z 90.100} C_DIS
   LIN {X -6.253, Y -19.953, Z 90.100} C_DIS
   LIN {X -5.709, Y -22.400, Z 90.100} C_DIS
   LIN {X -4.447, Y -24.283, Z 90.100} C_DIS
   LIN {X -4.089, Y -24.821, Z 90.100} C_DIS
   LIN {X -3.775, Y -25.062, Z 90.100} C_DIS
   LIN {X -1.328, Y -26.799, Z 90.100} C_DIS
   LIN {X 0.505, Y -27.259, Z 90.100} C_DIS
   LIN {X 3.411, Y -27.192, Z 90.100} C_DIS
   LIN {X 5.286, Y -27.177, Z 90.100} C_DIS
   LIN {X 6.489, Y -26.570, Z 90.100} C_DIS
   LIN {X 8.177, Y -25.593, Z 90.100} C_DIS
   LIN {X 10.035, Y -23.396, Z 90.100} C_DIS
   LIN {X 10.398, Y -22.916, Z 90.100} C_DIS
   LIN {X 10.645, Y -22.057, Z 90.100} C_DIS
   LIN {X 11.492, Y -19.362, Z 90.100} C_DIS
   LIN {X 11.639, Y -17.436, Z 90.100} C_DIS
   LIN {X 11.733, Y -16.109, Z 90.100} C_DIS
   LIN {X 11.817, Y -14.242, Z 90.100} C_DIS
   LIN {X 11.871, Y -13.152, Z 90.100} C_DIS
   LIN {X 11.888, Y -12.328, Z 90.100} C_DIS
   LIN {X 11.931, Y -9.348, Z 90.100} C_DIS
   LIN {X 11.877, Y -6.642, Z 90.100} C_DIS
   LIN {X 11.821, Y -4.563, Z 90.100} C_DIS
   LIN {X 11.629, Y -2.190, Z 90.100} C_DIS
   LIN {X 11.443, Y 0.103, Z 90.100} C_DIS
   LIN {X 11.384, Y 0.834, Z 90.100} C_DIS
   LIN {X 11.316, Y 2.143, Z 90.100} C_DIS
   LIN {X 10.962, Y 4.684, Z 90.100} C_DIS
   LIN {X 9.738, Y 12.481, Z 90.100} C_DIS
   LIN {X 7.782, Y 20.157, Z 90.100} C_DIS
   LIN {X 7.356, Y 21.960, Z 90.100} C_DIS
   LIN {X 5.947, Y 26.147, Z 90.100}
   LaserEnd_Ext()
   LIN {X -3.518, Y 44.522, Z 90.100}
   LaserStart_Ext()
   LIN {X -7.297, Y 44.522, Z 90.100}
   LaserEnd_Ext()
   LIN {X -8.239, Y 43.522, Z 90.100}
   LaserStart_Ext()
   LIN {X -2.758, Y 43.522, Z 90.100}
   LaserEnd_Ext()
   LIN {X -2.214, Y 42.522, Z 90.100}
   LaserStart_Ext()
   LIN {X -8.490, Y 42.522, Z 90.100}
   LaserEnd_Ext()
   LIN {X -8.327, Y 41.522, Z 90.100}
   LaserStart_Ext()
   LIN {X -1.686, Y 41.522, Z 90.100}
   LaserEnd_Ext()
   LIN {X -1.167, Y 40.522, Z 90.100}
   LaserStart_Ext()
   LIN {X -7.952, Y 40.522, Z 90.100}
   LaserEnd_Ext()
   LIN {X -7.491, Y 39.522, Z 90.100}
   LaserStart_Ext()
   LIN {X -0.665, Y 39.522, Z 90.100}
   LaserEnd_Ext()
   LIN {X -0.166, Y 38.522, Z 90.100}
   LaserStart_Ext()
   LIN {X -7.039, Y 38.522, Z 90.100}
   LaserEnd_Ext()
   LIN {X -6.618, Y 37.522, Z 90.100}
   LaserStart_Ext()
   LIN {X 0.298, Y 37.522, Z 90.100}
   LaserEnd_Ext()
   LIN {X 0.757, Y 36.522, Z 90.100}
   LaserStart_Ext()
   LIN {X -6.198, Y 36.522, Z 90.100}
   LaserEnd_Ext()
   LIN {X -5.811, Y 35.522, Z 90.100}
   LaserStart_Ext()
   LIN {X 1.216, Y 35.522, Z 90.100}
   LaserEnd_Ext()
   LIN {X 1.678, Y 34.522, Z 90.100}
   LaserStart_Ext()
   LIN {X -5.431, Y 34.522, Z 90.100}
   LaserEnd_Ext()
   LIN {X -5.057, Y 33.522, Z 90.100}
   LaserStart_Ext()
   LIN {X 2.106, Y 33.522, Z 90.100}
   LaserEnd_Ext()
   LIN {X 2.516, Y 32.522, Z 90.100}
   LaserStart_Ext()
   LIN {X -4.720, Y 32.522, Z 90.100}
   LaserEnd_Ext()
   LIN {X -4.388, Y 31.522, Z 90.100}
   LaserStart_Ext()
   LIN {X 2.926, Y 31.522, Z 90.100}
   LaserEnd_Ext()
   LIN {X 3.336, Y 30.522, Z 90.100}
   LaserStart_Ext()
   LIN {X -4.072, Y 30.522, Z 90.100}
   LaserEnd_Ext()
   LIN {X -3.773, Y 29.522, Z 90.100}
   LaserStart_Ext()
   LIN {X 3.712, Y 29.522, Z 90.100}
   LaserEnd_Ext()
   LIN {X 4.060, Y 28.522, Z 90.100}
   LaserStart_Ext()
   LIN {X -3.486, Y 28.522, Z 90.100}
   LaserEnd_Ext()
   LIN {X -3.215, Y 27.522, Z 90.100}
   LaserStart_Ext()
   LIN {X 4.409, Y 27.522, Z 90.100}
   LaserEnd_Ext()
   LIN {X 4.758, Y 26.522, Z 90.100}
   LaserStart_Ext()
   LIN {X -2.989, Y 26.522, Z 90.100}
   LaserEnd_Ext()
   LIN {X -2.763, Y 25.522, Z 90.100}
   LaserStart_Ext()
   LIN {X 5.102, Y 25.522, Z 90.100}
   LaserEnd_Ext()
   LIN {X 5.439, Y 24.522, Z 90.100}
   LaserStart_Ext()
   LIN {X -2.537, Y 24.522, Z 90.100}
   LaserEnd_Ext()
   LIN {X -2.339, Y 23.522, Z 90.100}
   LaserStart_Ext()
   LIN {X 5.775, Y 23.522, Z 90.100}
   LaserEnd_Ext()
   LIN {X 6.111, Y 22.522, Z 90.100}
   LaserStart_Ext()
   LIN {X -2.194, Y 22.522, Z 90.100}
   LaserEnd_Ext()
   LIN {X -2.050, Y 21.522, Z 90.100}
   LaserStart_Ext()
   LIN {X 6.431, Y 21.522, Z 90.100}
   LaserEnd_Ext()
   LIN {X 6.668, Y 20.522, Z 90.100}
   LaserStart_Ext()
   LIN {X -1.905, Y 20.522, Z 90.100}
   LaserEnd_Ext()
   LIN {X -1.761, Y 19.522, Z 90.100}
   LaserStart_Ext()
   LIN {X 6.912, Y 19.522, Z 90.100}
   LaserEnd_Ext()
   LIN {X 7.167, Y 18.522, Z 90.100}
   LaserStart_Ext()
   LIN {X -1.617, Y 18.522, Z 90.100}
   LaserEnd_Ext()
   LIN {X -1.472, Y 17.522, Z 90.100}
   LaserStart_Ext()
   LIN {X 7.421, Y 17.522, Z 90.100}
   LaserEnd_Ext()
   LIN {X 7.676, Y 16.522, Z 90.100}
   LaserStart_Ext()
   LIN {X -1.328, Y 16.522, Z 90.100}
   LaserEnd_Ext()
   LIN {X -1.184, Y 15.522, Z 90.100}
   LaserStart_Ext()
   LIN {X 7.931, Y 15.522, Z 90.100}
   LaserEnd_Ext()
   LIN {X 8.186, Y 14.522, Z 90.100}
   LaserStart_Ext()
   LIN {X -1.044, Y 14.522, Z 90.100}
   LaserEnd_Ext()
   LIN {X -0.953, Y 13.522, Z 90.100}
   LaserStart_Ext()
   LIN {X 8.441, Y 13.522, Z 90.100}
   LaserEnd_Ext()
   LIN {X 8.696, Y 12.522, Z 90.100}
   LaserStart_Ext()
   LIN {X -0.903, Y 12.522, Z 90.100}
   LaserEnd_Ext()
   LIN {X -0.901, Y 11.522, Z 90.100}
   LaserStart_Ext()
   LIN {X 8.876, Y 11.522, Z 90.100}
   LaserEnd_Ext()
   LIN {X 9.033, Y 10.522, Z 90.100}
   LaserStart_Ext()
   LIN {X -0.899, Y 10.522, Z 90.100}
   LaserEnd_Ext()
   LIN {X -0.896, Y 9.522, Z 90.100}
   LaserStart_Ext()
   LIN {X 9.190, Y 9.522, Z 90.100}
   LaserEnd_Ext()
   LIN {X 9.347, Y 8.522, Z 90.100}
   LaserStart_Ext()
   LIN {X -0.894, Y 8.522, Z 90.100}
   LaserEnd_Ext()
   LIN {X -0.892, Y 7.522, Z 90.100}
   LaserStart_Ext()
   LIN {X 9.504, Y 7.522, Z 90.100}
   LaserEnd_Ext()
   LIN {X 9.661, Y 6.522, Z 90.100}
   LaserStart_Ext()
   LIN {X -0.890, Y 6.522, Z 90.100}
   LaserEnd_Ext()
   LIN {X -0.888, Y 5.522, Z 90.100}
   LaserStart_Ext()
   LIN {X 9.818, Y 5.522, Z 90.100}
   LaserEnd_Ext()
   LIN {X 9.975, Y 4.522, Z 90.100}
   LaserStart_Ext()
   LIN {X -0.895, Y 4.522, Z 90.100}
   LaserEnd_Ext()
   LIN {X -0.986, Y 3.522, Z 90.100}
   LaserStart_Ext()
   LIN {X 10.114, Y 3.522, Z 90.100}
   LaserEnd_Ext()
   LIN {X 10.253, Y 2.522, Z 90.100}
   LaserStart_Ext()
   LIN {X -1.081, Y 2.522, Z 90.100}
   LaserEnd_Ext()
   LIN {X -1.174, Y 1.522, Z 90.100}
   LaserStart_Ext()
   LIN {X 10.347, Y 1.522, Z 90.100}
   LaserEnd_Ext()
   LIN {X 10.406, Y 0.522, Z 90.100}
   LaserStart_Ext()
   LIN {X -1.267, Y 0.522, Z 90.100}
   LaserEnd_Ext()
   LIN {X -1.360, Y -0.478, Z 90.100}
   LaserStart_Ext()
   LIN {X 10.487, Y -0.478, Z 90.100}
   LaserEnd_Ext()
   LIN {X 10.568, Y -1.478, Z 90.100}
   LaserStart_Ext()
   LIN {X -1.491, Y -1.478, Z 90.100}
   LaserEnd_Ext()
   LIN {X -1.643, Y -2.478, Z 90.100}
   LaserStart_Ext()
   LIN {X 10.649, Y -2.478, Z 90.100}
   LaserEnd_Ext()
   LIN {X 10.730, Y -3.478, Z 90.100}
   LaserStart_Ext()
   LIN {X -1.795, Y -3.478, Z 90.100}
   LaserEnd_Ext()
   LIN {X -1.980, Y -4.478, Z 90.100}
   LaserStart_Ext()
   LIN {X 10.811, Y -4.478, Z 90.100}
   LaserEnd_Ext()
   LIN {X 10.845, Y -5.478, Z 90.100}
   LaserStart_Ext()
   LIN {X -2.172, Y -5.478, Z 90.100}
   LaserEnd_Ext()
   LIN {X -2.364, Y -6.478, Z 90.100}
   LaserStart_Ext()
   LIN {X 10.872, Y -6.478, Z 90.100}
   LaserEnd_Ext()
   LIN {X 10.894, Y -7.478, Z 90.100}
   LaserStart_Ext()
   LIN {X -2.590, Y -7.478, Z 90.100}
   LaserEnd_Ext()
   LIN {X -2.826, Y -8.478, Z 90.100}
   LaserStart_Ext()
   LIN {X 10.914, Y -8.478, Z 90.100}
   LaserEnd_Ext()
   LIN {X 10.929, Y -9.478, Z 90.100}
   LaserStart_Ext()
   LIN {X -3.063, Y -9.478, Z 90.100}
   LaserEnd_Ext()
   LIN {X -3.333, Y -10.478, Z 90.100}
   LaserStart_Ext()
   LIN {X 10.915, Y -10.478, Z 90.100}
   LaserEnd_Ext()
   LIN {X 10.900, Y -11.478, Z 90.100}
   LaserStart_Ext()
   LIN {X -3.618, Y -11.478, Z 90.100}
   LaserEnd_Ext()
   LIN {X -3.902, Y -12.478, Z 90.100}
   LaserStart_Ext()
   LIN {X 10.885, Y -12.478, Z 90.100}
   LaserEnd_Ext()
   LIN {X 10.853, Y -13.478, Z 90.100}
   LaserStart_Ext()
   LIN {X 5.430, Y -13.478, Z 90.100}
   LaserEnd_Ext()
   LIN {X -0.317, Y -13.478, Z 90.100}
   LaserStart_Ext()
   LIN {X -4.210, Y -13.478, Z 90.100}
   LaserEnd_Ext()
   LIN {X -4.542, Y -14.478, Z 90.100}
   LaserStart_Ext()
   LIN {X -1.699, Y -14.478, Z 90.100}
   LaserEnd_Ext()
   LIN {X 6.723, Y -14.478, Z 90.100}
   LaserStart_Ext()
   LIN {X 10.805, Y -14.478, Z 90.100}
   LaserEnd_Ext()
   LIN {X 10.760, Y -15.478, Z 90.100}
   LaserStart_Ext()
   LIN {X 7.469, Y -15.478, Z 90.100}
   LaserEnd_Ext()
   LIN {X -2.551, Y -15.478, Z 90.100}
   LaserStart_Ext()
   LIN {X -4.873, Y -15.478, Z 90.100}
   LaserEnd_Ext()
   LIN {X -5.108, Y -16.478, Z 90.100}
   LaserStart_Ext()
   LIN {X -2.952, Y -16.478, Z 90.100}
   LaserEnd_Ext()
   LIN {X 8.123, Y -16.478, Z 90.100}
   LaserStart_Ext()
   LIN {X 10.704, Y -16.478, Z 90.100}
   LaserEnd_Ext()
   LIN {X 10.633, Y -17.478, Z 90.100}
   LaserStart_Ext()
   LIN {X 8.287, Y -17.478, Z 90.100}
   LaserEnd_Ext()
   LIN {X -3.177, Y -17.478, Z 90.100}
   LaserStart_Ext()
   LIN {X -5.275, Y -17.478, Z 90.100}
   LaserEnd_Ext()
   LIN {X -5.443, Y -18.478, Z 90.100}
   LaserStart_Ext()
   LIN {X -3.402, Y -18.478, Z 90.100}
   LaserEnd_Ext()
   LIN {X 8.445, Y -18.478, Z 90.100}
   LaserStart_Ext()
   LIN {X 10.557, Y -18.478, Z 90.100}
   LaserEnd_Ext()
   LIN {X 10.407, Y -19.478, Z 90.100}
   LaserStart_Ext()
   LIN {X 8.375, Y -19.478, Z 90.100}
   LaserEnd_Ext()
   LIN {X -3.388, Y -19.478, Z 90.100}
   LaserStart_Ext()
   LIN {X -5.333, Y -19.478, Z 90.100}
   LaserEnd_Ext()
   LIN {X -5.112, Y -20.478, Z 90.100}
   LaserStart_Ext()
   LIN {X -3.109, Y -20.478, Z 90.100}
   LaserEnd_Ext()
   LIN {X 8.072, Y -20.478, Z 90.100}
   LaserStart_Ext()
   LIN {X 10.093, Y -20.478, Z 90.100}
   LaserEnd_Ext()
   LIN {X 9.779, Y -21.478, Z 90.100}
   LaserStart_Ext()
   LIN {X 7.763, Y -21.478, Z 90.100}
   LaserEnd_Ext()
   LIN {X -2.799, Y -21.478, Z 90.100}
   LaserStart_Ext()
   LIN {X -4.890, Y -21.478, Z 90.100}
   LaserEnd_Ext()
   LIN {X -4.453, Y -22.478, Z 90.100}
   LaserStart_Ext()
   LIN {X -1.982, Y -22.478, Z 90.100}
   LaserEnd_Ext()
   LIN {X 6.936, Y -22.478, Z 90.100}
   LaserStart_Ext()
   LIN {X 9.475, Y -22.478, Z 90.100}
   LaserEnd_Ext()
   LIN {X 8.655, Y -23.478, Z 90.100}
   LaserStart_Ext()
   LIN {X 6.011, Y -23.478, Z 90.100}
   LaserEnd_Ext()
   LIN {X -1.030, Y -23.478, Z 90.100}
   LaserStart_Ext()
   LIN {X -3.783, Y -23.478, Z 90.100}
   LaserEnd_Ext()
   LIN {X -2.870, Y -24.478, Z 90.100}
   LaserStart_Ext()
   LIN {X 1.130, Y -24.478, Z 90.100}
   LaserEnd_Ext()
   LIN {X 3.728, Y -24.478, Z 90.100}
   LaserStart_Ext()
   LIN {X 7.809, Y -24.478, Z 90.100}
   LaserEnd_Ext()
   LIN {X 6.379, Y -25.478, Z 90.100}
   LaserStart_Ext()
   LIN {X -1.461, Y -25.478, Z 90.100}
   LaserEnd_Ext()
   LIN {X -1.556, Y -21.282, Z 90.950}
   LaserStart_Ext()
   LIN {X -1.842, Y -20.941, Z 90.950} C_DIS
   LIN {X -1.961, Y -20.516, Z 90.950} C_DIS
   LIN {X -2.408, Y -18.933, Z 90.950} C_DIS
   LIN {X -1.773, Y -16.137, Z 90.950} C_DIS
   LIN {X -0.434, Y -14.591, Z 90.950} C_DIS
   LIN {X 0.893, Y -14.010, Z 90.950} C_DIS
   LIN {X 1.728, Y -13.640, Z 90.950} C_DIS
   LIN {X 2.947, Y -13.668, Z 90.950} C_DIS
   LIN {X 3.800, Y -13.695, Z 90.950} C_DIS
   LIN {X 4.417, Y -13.999, Z 90.950} C_DIS
   LIN {X 5.708, Y -14.630, Z 90.950} C_DIS
   LIN {X 6.773, Y -16.048, Z 90.950} C_DIS
   LIN {X 7.233, Y -16.665, Z 90.950} C_DIS
   LIN {X 7.353, Y -17.420, Z 90.950} C_DIS
   LIN {X 7.583, Y -18.847, Z 90.950} C_DIS
   LIN {X 7.141, Y -20.315, Z 90.950} C_DIS
   LIN {X 6.922, Y -21.035, Z 90.950} C_DIS
   LIN {X 6.293, Y -21.730, Z 90.950} C_DIS
   LIN {X 5.469, Y -22.642, Z 90.950} C_DIS
   LIN {X 4.803, Y -22.923, Z 90.950} C_DIS
   LIN {X 3.455, Y -23.489, Z 90.950} C_DIS
   LIN {X 1.428, Y -23.436, Z 90.950} C_DIS
   LIN {X 1.279, Y -23.394, Z 90.950} C_DIS
   LIN {X -0.497, Y -22.532, Z 90.950} C_DIS
   LIN {X -1.556, Y -21.282, Z 90.950}
   LaserEnd_Ext()
   LIN {X -3.069, Y 45.505, Z 90.950}
   LaserStart_Ext()
   LIN {X -4.127, Y 46.052, Z 90.950} C_DIS
   LIN {X -4.614, Y 46.301, Z 90.950} C_DIS
   LIN {X -5.496, Y 46.333, Z 90.950} C_DIS
   LIN {X -6.358, Y 46.366, Z 90.950} C_DIS
   LIN {X -7.101, Y 45.903, Z 90.950} C_DIS
   LIN {X -8.819, Y 44.824, Z 90.950} C_DIS
   LIN {X -9.452, Y 43.393, Z 90.950} C_DIS
   LIN {X -9.527, Y 43.230, Z 90.950} C_DIS
   LIN {X -9.534, Y 43.030, Z 90.950} C_DIS
   LIN {X -9.568, Y 41.965, Z 90.950} C_DIS
   LIN {X -9.231, Y 40.845, Z 90.950} C_DIS
   LIN {X -9.185, Y 40.700, Z 90.950} C_DIS
   LIN {X -9.135, Y 40.596, Z 90.950} C_DIS
   LIN {X -8.652, Y 39.569, Z 90.950} C_DIS
   LIN {X -8.107, Y 38.371, Z 90.950} C_DIS
   LIN {X -7.990, Y 38.113, Z 90.950} C_DIS
   LIN {X -7.814, Y 37.693, Z 90.950} C_DIS
   LIN {X -7.068, Y 35.929, Z 90.950} C_DIS
   LIN {X -6.424, Y 34.245, Z 90.950} C_DIS
   LIN {X -6.086, Y 33.355, Z 90.950} C_DIS
   LIN {X -5.171, Y 30.638, Z 90.950} C_DIS
   LIN {X -5.026, Y 30.179, Z 90.950} C_DIS
   LIN {X -4.163, Y 27.166, Z 90.950} C_DIS
   LIN {X -3.464, Y 24.075, Z 90.950} C_DIS
   LIN {X -1.919, Y 13.371, Z 90.950} C_DIS
   LIN {X -1.902, Y 13.255, Z 90.950} C_DIS
   LIN {X -1.869, Y 4.720, Z 90.950} C_DIS
   LIN {X -1.885, Y 4.300, Z 90.950} C_DIS
   LIN {X -2.336, Y -0.548, Z 90.950} C_DIS
   LIN {X -2.390, Y -0.975, Z 90.950} C_DIS
   LIN {X -2.665, Y -2.782, Z 90.950} C_DIS
   LIN {X -2.791, Y -3.617, Z 90.950} C_DIS
   LIN {X -3.323, Y -6.374, Z 90.950} C_DIS
   LIN {X -3.375, Y -6.648, Z 90.950} C_DIS
   LIN {X -3.400, Y -6.753, Z 90.950} C_DIS
   LIN {X -4.079, Y -9.625, Z 90.950} C_DIS
   LIN {X -4.654, Y -11.652, Z 90.950} C_DIS
   LIN {X -4.957, Y -12.727, Z 90.950} C_DIS
   LIN {X -5.240, Y -13.593, Z 90.950} C_DIS
   LIN {X -5.910, Y -15.614, Z 90.950} C_DIS
   LIN {X -6.325, Y -18.106, Z 90.950} C_DIS
   LIN {X -6.428, Y -18.742, Z 90.950} C_DIS
   LIN {X -6.275, Y -19.413, Z 90.950} C_DIS
   LIN {X -5.619, Y -22.363, Z 90.950} C_DIS
   LIN {X -4.431, Y -24.134, Z 90.950} C_DIS
   LIN {X -3.990, Y -24.783, Z 90.950} C_DIS
   LIN {X -2.943, Y -25.493, Z 90.950} C_DIS
   LIN {X -1.060, Y -26.829, Z 90.950} C_DIS
   LIN {X -0.027, Y -27.088, Z 90.950} C_DIS
   LIN {X 1.610, Y -27.050, Z 90.950} C_DIS
   LIN {X 5.671, Y -27.018, Z 90.950} C_DIS
   LIN {X 5.787, Y -26.959, Z 90.950} C_DIS
   LIN {X 8.288, Y -25.511, Z 90.950} C_DIS
   LIN {X 9.568, Y -23.997, Z 90.950} C_DIS
   LIN {X 10.575, Y -22.667, Z 90.950} C_DIS
   LIN {X 11.260, Y -20.286, Z 90.950} C_DIS
   LIN {X 11.575, Y -19.284, Z 90.950} C_DIS
   LIN {X 11.630, Y -18.568, Z 90.950} C_DIS
   LIN {X 11.808, Y -16.030, Z 90.950} C_DIS
   LIN {X 11.921, Y -13.524, Z 90.950} C_DIS
   LIN {X 11.939, Y -13.072, Z 90.950} C_DIS
   LIN {X 11.956, Y -11.707, Z 90.950} C_DIS
   LIN {X 11.991, Y -9.269, Z 90.950} C_DIS
   LIN {X 11.969, Y -8.210, Z 90.950} C_DIS
   LIN {X 11.869, Y -4.484, Z 90.950} C_DIS
   LIN {X 11.525, Y -0.230, Z 90.950} C_DIS
   LIN {X 11.419, Y 1.075, Z 90.950} C_DIS
   LIN {X 11.385, Y 1.492, Z 90.950} C_DIS
   LIN {X 11.346, Y 2.237, Z 90.950} C_DIS
   LIN {X 11.145, Y 3.685, Z 90.950} C_DIS
   LIN {X 9.778, Y 12.395, Z 90.950} C_DIS
   LIN {X 7.592, Y 20.969, Z 90.950} C_DIS
   LIN {X 7.351, Y 21.989, Z 90.950} C_DIS
   LIN {X 6.554, Y 24.359, Z 90.950} C_DIS
   LIN {X 4.398, Y 30.544, Z 90.950} C_DIS
   LIN {X 2.898, Y 34.205, Z 90.950} C_DIS
   LIN {X 2.138, Y 35.856, Z 90.950} C_DIS
   LIN {X 1.957, Y 36.246, Z 90.950} C_DIS
   LIN {X 1.569, Y 37.083, Z 90.950} C_DIS
   LIN {X 0.734, Y 38.901, Z 90.950} C_DIS
   LIN {X 0.005, Y 40.345, Z 90.950} C_DIS
   LIN {X -0.516, Y 41.381, Z 90.950} C_DIS
   LIN {X -0.747, Y 41.819, Z 90.950} C_DIS
   LIN {X -1.414, Y 43.074, Z 90.950} C_DIS
   LIN {X -2.102, Y 44.333, Z 90.950} C_DIS
   LIN {X -3.069, Y 45.505, Z 90.950}
   LaserEnd_Ext()
   LIN {X -8.280, Y 43.570, Z 90.950}
   LaserStart_Ext()
   LIN {X -8.280, Y 41.156, Z 90.950}
   LaserEnd_Ext()
   LIN {X -7.280, Y 38.968, Z 90.950}
   LaserStart_Ext()
   LIN {X -7.280, Y 44.610, Z 90.950}
   LaserEnd_Ext()
   LIN {X -6.280, Y 45.236, Z 90.950}
   LaserStart_Ext()
   LIN {X -6.280, Y 36.633, Z 90.950}
   LaserEnd_Ext()
   LIN {X -5.280, Y -19.281, Z 90.950}
   LaserStart_Ext()
   LIN {X -5.280, Y -17.917, Z 90.950}
   LaserEnd_Ext()
   LIN {X -5.280, Y 34.050, Z 90.950}
   LaserStart_Ext()
   LIN {X -5.280, Y 45.325, Z 90.950}
   LaserEnd_Ext()
   LIN {X -4.280, Y 45.005, Z 90.950}
   LaserStart_Ext()
   LIN {X -4.280, Y 31.126, Z 90.950}
   LaserEnd_Ext()
   LIN {X -4.280, Y -13.875, Z 90.950}
   LaserStart_Ext()
   LIN {X -4.280, Y -22.564, Z 90.950}
   LaserEnd_Ext()
   LIN {X -3.280, Y -24.049, Z 90.950}
   LaserStart_Ext()
   LIN {X -3.280, Y -19.527, Z 90.950}
   LaserEnd_Ext()
   LIN {X -3.280, Y -18.256, Z 90.950}
   LaserStart_Ext()
   LIN {X -3.280, Y -10.472, Z 90.950}
   LaserEnd_Ext()
   LIN {X -3.280, Y 27.715, Z 90.950}
   LaserStart_Ext()
   LIN {X -3.280, Y 44.198, Z 90.950}
   LaserEnd_Ext()
   LIN {X -2.280, Y 42.573, Z 90.950}
   LaserStart_Ext()
   LIN {X -2.280, Y 22.870, Z 90.950}
   LaserEnd_Ext()
   LIN {X -2.280, Y -6.247, Z 90.950}
   LaserStart_Ext()
   LIN {X -2.280, Y -15.194, Z 90.950}
   LaserEnd_Ext()
   LIN {X -2.280, Y -21.975, Z 90.950}
   LaserStart_Ext()
   LIN {X -2.280, Y -24.737, Z 90.950}
   LaserEnd_Ext()
   LIN {X -1.280, Y -25.446, Z 90.950}
   LaserStart_Ext()
   LIN {X -1.280, Y -23.155, Z 90.950}
   LaserEnd_Ext()
   LIN {X -1.280, Y -14.040, Z 90.950}
   LaserStart_Ext()
   LIN {X -1.280, Y 0.013, Z 90.950}
   LaserEnd_Ext()
   LIN {X -1.280, Y 15.943, Z 90.950}
   LaserStart_Ext()
   LIN {X -1.280, Y 40.675, Z 90.950}
   LaserEnd_Ext()
   LIN {X -0.280, Y 38.690, Z 90.950}
   LaserStart_Ext()
   LIN {X -0.280, Y -13.432, Z 90.950}
   LaserEnd_Ext()
   LIN {X -0.280, Y -23.749, Z 90.950}
   LaserStart_Ext()
   LIN {X -0.280, Y -25.993, Z 90.950}
   LaserEnd_Ext()
   LIN {X 0.720, Y -26.070, Z 90.950}
   LaserStart_Ext()
   LIN {X 0.720, Y -24.234, Z 90.950}
   LaserEnd_Ext()
   LIN {X 0.720, Y -12.993, Z 90.950}
   LaserStart_Ext()
   LIN {X 0.720, Y 36.536, Z 90.950}
   LaserEnd_Ext()
   LIN {X 1.720, Y 34.372, Z 90.950}
   LaserStart_Ext()
   LIN {X 1.720, Y -12.642, Z 90.950}
   LaserEnd_Ext()
   LIN {X 1.720, Y -24.444, Z 90.950}
   LaserStart_Ext()
   LIN {X 1.720, Y -26.049, Z 90.950}
   LaserEnd_Ext()
   LIN {X 2.720, Y -26.041, Z 90.950}
   LaserStart_Ext()
   LIN {X 2.720, Y -24.470, Z 90.950}
   LaserEnd_Ext()
   LIN {X 2.720, Y -12.663, Z 90.950}
   LaserStart_Ext()
   LIN {X 2.720, Y 32.001, Z 90.950}
   LaserEnd_Ext()
   LIN {X 3.720, Y 29.451, Z 90.950}
   LaserStart_Ext()
   LIN {X 3.720, Y -12.692, Z 90.950}
   LaserEnd_Ext()
   LIN {X 3.720, Y -24.453, Z 90.950}
   LaserStart_Ext()
   LIN {X 3.720, Y -26.033, Z 90.950}
   LaserEnd_Ext()
   LIN {X 4.720, Y -26.025, Z 90.950}
   LaserStart_Ext()
   LIN {X 4.720, Y -24.043, Z 90.950}
   LaserEnd_Ext()
   LIN {X 4.720, Y -13.034, Z 90.950}
   LaserStart_Ext()
   LIN {X 4.720, Y 26.582, Z 90.950}
   LaserEnd_Ext()
   LIN {X 5.720, Y 23.702, Z 90.950}
   LaserStart_Ext()
   LIN {X 5.720, Y -13.523, Z 90.950}
   LaserEnd_Ext()
   LIN {X 5.720, Y -23.621, Z 90.950}
   LaserStart_Ext()
   LIN {X 5.720, Y -25.842, Z 90.950}
   LaserEnd_Ext()
   LIN {X 6.720, Y -25.263, Z 90.950}
   LaserStart_Ext()
   LIN {X 6.720, Y -22.749, Z 90.950}
   LaserEnd_Ext()
   LIN {X 6.720, Y -14.312, Z 90.950}
   LaserStart_Ext()
   LIN {X 6.720, Y 20.342, Z 90.950}
   LaserEnd_Ext()
   LIN {X 7.720, Y 16.418, Z 90.950}
   LaserStart_Ext()
   LIN {X 7.720, Y -15.645, Z 90.950}
   LaserEnd_Ext()
   LIN {X 7.720, Y -21.636, Z 90.950}
   LaserStart_Ext()
   LIN {X 7.720, Y -24.634, Z 90.950}
   LaserEnd_Ext()
   LIN {X 8.720, Y -23.452, Z 90.950}
   LaserStart_Ext()
   LIN {X 8.720, Y 12.495, Z 90.950}
   LaserEnd_Ext()
   LIN {X 9.720, Y 6.312, Z 90.950}
   LaserStart_Ext()
   LIN {X 9.720, Y -22.021, Z 90.950}
   LaserEnd_Ext()
   LIN {X 10.720, Y -17.247, Z 90.950}
   LaserStart_Ext()
   LIN {X 10.720, Y -2.685, Z 90.950}
   LaserEnd_Ext()
   LIN {X 3.870, Y -13.635, Z 91.800}
   LaserStart_Ext()
   LIN {X 4.546, Y -13.962, Z 91.800} C_DIS
   LIN {X 5.780, Y -14.565, Z 91.800} C_DIS
   LIN {X 6.734, Y -15.835, Z 91.800} C_DIS
   LIN {X 7.310, Y -16.597, Z 91.800} C_DIS
   LIN {X 7.429, Y -17.318, Z 91.800} C_DIS
   LIN {X 7.665, Y -18.778, Z 91.800} C_DIS
   LIN {X 7.231, Y -20.216, Z 91.800} C_DIS
   LIN {X 7.024, Y -20.940, Z 91.800} C_DIS
   LIN {X 6.541, Y -21.490, Z 91.800} C_DIS
   LIN {X 5.553, Y -22.582, Z 91.800} C_DIS
   LIN {X 3.722, Y -23.357, Z 91.800} C_DIS
   LIN {X 3.548, Y -23.430, Z 91.800} C_DIS
   LIN {X 3.265, Y -23.423, Z 91.800} C_DIS
   LIN {X 1.455, Y -23.380, Z 91.800} C_DIS
   LIN {X 0.300, Y -22.825, Z 91.800} C_DIS
   LIN {X -0.407, Y -22.482, Z 91.800} C_DIS
   LIN {X -1.021, Y -21.757, Z 91.800} C_DIS
   LIN {X -1.756, Y -20.895, Z 91.800} C_DIS
   LIN {X -2.042, Y -19.894, Z 91.800} C_DIS
   LIN {X -2.326, Y -18.888, Z 91.800} C_DIS
   LIN {X -2.066, Y -17.740, Z 91.800} C_DIS
   LIN {X -1.694, Y -16.083, Z 91.800} C_DIS
   LIN {X -0.412, Y -14.612, Z 91.800} C_DIS
   LIN {X -0.326, Y -14.513, Z 91.800} C_DIS
   LIN {X 1.755, Y -13.593, Z 91.800} C_DIS
   LIN {X 3.245, Y -13.627, Z 91.800} C_DIS
   LIN {X 3.870, Y -13.635, Z 91.800}
   LaserEnd_Ext()
   LIN {X -6.886, Y 35.364, Z 91.800}
   LaserStart_Ext()
   LIN {X -6.128, Y 33.395, Z 91.800} C_DIS
   LIN {X -5.418, Y 31.286, Z 91.800} C_DIS
   LIN {X -5.260, Y 30.817, Z 91.800} C_DIS
   LIN {X -5.091, Y 30.329, Z 91.800} C_DIS
   LIN {X -4.877, Y 29.573, Z 91.800} C_DIS
   LIN {X -4.084, Y 26.805, Z 91.800} C_DIS
   LIN {X -3.557, Y 24.474, Z 91.800} C_DIS
   LIN {X -2.391, Y 16.399, Z 91.800} C_DIS
   LIN {X -1.955, Y 13.780, Z 91.800} C_DIS
   LIN {X -1.871, Y 12.895, Z 91.800} C_DIS
   LIN {X -1.842, Y 5.071, Z 91.800} C_DIS
   LIN {X -1.883, Y 3.941, Z 91.800} C_DIS
   LIN {X -2.296, Y -0.484, Z 91.800} C_DIS
   LIN {X -2.374, Y -1.105, Z 91.800} C_DIS
   LIN {X -2.546, Y -2.237, Z 91.800} C_DIS
   LIN {X -2.775, Y -3.748, Z 91.800} C_DIS
   LIN {X -3.213, Y -6.022, Z 91.800} C_DIS
   LIN {X -3.423, Y -7.063, Z 91.800} C_DIS
   LIN {X -3.940, Y -9.232, Z 91.800} C_DIS
   LIN {X -4.062, Y -9.748, Z 91.800} C_DIS
   LIN {X -4.151, Y -10.063, Z 91.800} C_DIS
   LIN {X -4.896, Y -12.711, Z 91.800} C_DIS
   LIN {X -5.593, Y -14.843, Z 91.800} C_DIS
   LIN {X -5.836, Y -15.577, Z 91.800} C_DIS
   LIN {X -5.987, Y -16.482, Z 91.800} C_DIS
   LIN {X -6.346, Y -18.706, Z 91.800} C_DIS
   LIN {X -5.811, Y -21.054, Z 91.800} C_DIS
   LIN {X -5.528, Y -22.325, Z 91.800} C_DIS
   LIN {X -5.017, Y -23.088, Z 91.800} C_DIS
   LIN {X -3.890, Y -24.745, Z 91.800} C_DIS
   LIN {X -1.215, Y -26.558, Z 91.800} C_DIS
   LIN {X -0.792, Y -26.858, Z 91.800} C_DIS
   LIN {X -0.560, Y -26.917, Z 91.800} C_DIS
   LIN {X -0.192, Y -26.908, Z 91.800} C_DIS
   LIN {X 0.859, Y -26.900, Z 91.800} C_DIS
   LIN {X 5.668, Y -26.988, Z 91.800} C_DIS
   LIN {X 6.910, Y -26.292, Z 91.800} C_DIS
   LIN {X 8.400, Y -25.429, Z 91.800} C_DIS
   LIN {X 9.102, Y -24.599, Z 91.800} C_DIS
   LIN {X 10.752, Y -22.418, Z 91.800} C_DIS
   LIN {X 11.536, Y -19.694, Z 91.800} C_DIS
   LIN {X 11.658, Y -19.205, Z 91.800} C_DIS
   LIN {X 11.721, Y -18.262, Z 91.800} C_DIS
   LIN {X 11.884, Y -15.950, Z 91.800} C_DIS
   LIN {X 11.940, Y -14.698, Z 91.800} C_DIS
   LIN {X 12.008, Y -12.993, Z 91.800} C_DIS
   LIN {X 12.048, Y -9.650, Z 91.800} C_DIS
   LIN {X 12.050, Y -9.190, Z 91.800} C_DIS
   LIN {X 12.007, Y -7.758, Z 91.800} C_DIS
   LIN {X 11.917, Y -4.405, Z 91.800} C_DIS
   LIN {X 11.420, Y 1.729, Z 91.800} C_DIS
   LIN {X 11.395, Y 2.048, Z 91.800} C_DIS
   LIN {X 11.386, Y 2.150, Z 91.800} C_DIS
   LIN {X 11.377, Y 2.332, Z 91.800} C_DIS
   LIN {X 11.328, Y 2.686, Z 91.800} C_DIS
   LIN {X 9.817, Y 12.308, Z 91.800} C_DIS
   LIN {X 7.403, Y 21.782, Z 91.800} C_DIS
   LIN {X 7.347, Y 22.019, Z 91.800} C_DIS
   LIN {X 7.161, Y 22.571, Z 91.800} C_DIS
   LIN {X 4.341, Y 30.661, Z 91.800} C_DIS
   LIN {X 3.035, Y 33.847, Z 91.800} C_DIS
   LIN {X 1.872, Y 36.375, Z 91.800} C_DIS
   LIN {X 1.594, Y 36.972, Z 91.800} C_DIS
   LIN {X 1.001, Y 38.254, Z 91.800} C_DIS
   LIN {X 0.676, Y 38.961, Z 91.800} C_DIS
   LIN {X 0.077, Y 40.147, Z 91.800} C_DIS
   LIN {X -0.579, Y 41.436, Z 91.800} C_DIS
   LIN {X -1.349, Y 42.879, Z 91.800} C_DIS
   LIN {X -1.478, Y 43.121, Z 91.800} C_DIS
   LIN {X -1.554, Y 43.261, Z 91.800} C_DIS
   LIN {X -2.192, Y 44.422, Z 91.800} C_DIS
   LIN {X -2.977, Y 45.357, Z 91.800} C_DIS
   LIN {X -3.138, Y 45.549, Z 91.800} C_DIS
   LIN {X -3.492, Y 45.729, Z 91.800} C_DIS
   LIN {X -4.686, Y 46.341, Z 91.800} C_DIS
   LIN {X -5.554, Y 46.373, Z 91.800} C_DIS
   LIN {X -6.430, Y 46.402, Z 91.800} C_DIS
   LIN {X -8.725, Y 44.955, Z 91.800} C_DIS
   LIN {X -8.851, Y 44.889, Z 91.800} C_DIS
   LIN {X -9.055, Y 44.499, Z 91.800} C_DIS
   LIN {X -9.559, Y 43.403, Z 91.800} C_DIS
   LIN {X -9.586, Y 42.657, Z 91.800} C_DIS
   LIN {X -9.625, Y 41.947, Z 91.800} C_DIS
   LIN {X -9.508, Y 41.562, Z 91.800} C_DIS
   LIN {X -9.243, Y 40.729, Z 91.800} C_DIS
   LIN {X -8.732, Y 39.649, Z 91.800} C_DIS
   LIN {X -8.689, Y 39.557, Z 91.800} C_DIS
   LIN {X -8.042, Y 38.144, Z 91.800} C_DIS
   LIN {X -7.284, Y 36.361, Z 91.800} C_DIS
   LIN {X -7.115, Y 35.963, Z 91.800} C_DIS
   LIN {X -6.886, Y 35.364, Z 91.800}
   LaserEnd_Ext()
   LIN {X -1.200, Y -25.360, Z 91.800}
   LaserStart_Ext()
   LIN {X 6.523, Y -25.360, Z 91.800}
   LaserEnd_Ext()
   LIN {X 7.994, Y -24.360, Z 91.800}
   LaserStart_Ext()
   LIN {X 3.913, Y -24.360, Z 91.800}
   LaserEnd_Ext()
   LIN {X 1.265, Y -24.360, Z 91.800}
   LaserStart_Ext()
   LIN {X -2.676, Y -24.360, Z 91.800}
   LaserEnd_Ext()
   LIN {X -3.623, Y -23.360, Z 91.800}
   LaserStart_Ext()
   LIN {X -0.882, Y -23.360, Z 91.800}
   LaserEnd_Ext()
   LIN {X 6.179, Y -23.360, Z 91.800}
   LaserStart_Ext()
   LIN {X 8.785, Y -23.360, Z 91.800}
   LaserEnd_Ext()
   LIN {X 9.541, Y -22.360, Z 91.800}
   LaserStart_Ext()
   LIN {X 7.102, Y -22.360, Z 91.800}
   LaserEnd_Ext()
   LIN {X -1.821, Y -22.360, Z 91.800}
   LaserStart_Ext()
   LIN {X -4.301, Y -22.360, Z 91.800}
   LaserEnd_Ext()
   LIN {X -4.719, Y -21.360, Z 91.800}
   LaserStart_Ext()
   LIN {X -2.640, Y -21.360, Z 91.800}
   LaserEnd_Ext()
   LIN {X 7.930, Y -21.360, Z 91.800}
   LaserStart_Ext()
   LIN {X 10.016, Y -21.360, Z 91.800}
   LaserEnd_Ext()
   LIN {X 10.303, Y -20.360, Z 91.800}
   LaserStart_Ext()
   LIN {X 8.232, Y -20.360, Z 91.800}
   LaserEnd_Ext()
   LIN {X -2.949, Y -20.360, Z 91.800}
   LaserStart_Ext()
   LIN {X -4.944, Y -20.360, Z 91.800}
   LaserEnd_Ext()
   LIN {X -5.171, Y -19.360, Z 91.800}
   LaserStart_Ext()
   LIN {X -3.232, Y -19.360, Z 91.800}
   LaserEnd_Ext()
   LIN {X 8.534, Y -19.360, Z 91.800}
   LaserStart_Ext()
   LIN {X 10.588, Y -19.360, Z 91.800}
   LaserEnd_Ext()
   LIN {X 10.712, Y -18.360, Z 91.800}
   LaserStart_Ext()
   LIN {X 8.610, Y -18.360, Z 91.800}
   LaserEnd_Ext()
   LIN {X -3.232, Y -18.360, Z 91.800}
   LaserStart_Ext()
   LIN {X -5.277, Y -18.360, Z 91.800}
   LaserEnd_Ext()
   LIN {X -5.116, Y -17.360, Z 91.800}
   LaserStart_Ext()
   LIN {X -3.005, Y -17.360, Z 91.800}
   LaserEnd_Ext()
   LIN {X 8.449, Y -17.360, Z 91.800}
   LaserStart_Ext()
   LIN {X 10.782, Y -17.360, Z 91.800}
   LaserEnd_Ext()
   LIN {X 10.852, Y -16.360, Z 91.800}
   LaserStart_Ext()
   LIN {X 8.281, Y -16.360, Z 91.800}
   LaserEnd_Ext()
   LIN {X -2.781, Y -16.360, Z 91.800}
   LaserStart_Ext()
   LIN {X -4.953, Y -16.360, Z 91.800}
   LaserEnd_Ext()
   LIN {X -4.710, Y -15.360, Z 91.800}
   LaserStart_Ext()
   LIN {X -2.391, Y -15.360, Z 91.800}
   LaserEnd_Ext()
   LIN {X 7.628, Y -15.360, Z 91.800}
   LaserStart_Ext()
   LIN {X 10.909, Y -15.360, Z 91.800}
   LaserEnd_Ext()
   LIN {X 10.953, Y -14.360, Z 91.800}
   LaserStart_Ext()
   LIN {X 6.877, Y -14.360, Z 91.800}
   LaserEnd_Ext()
   LIN {X -1.519, Y -14.360, Z 91.800}
   LaserStart_Ext()
   LIN {X -4.383, Y -14.360, Z 91.800}
   LaserEnd_Ext()
   LIN {X -4.057, Y -13.360, Z 91.800}
   LaserStart_Ext()
   LIN {X -0.190, Y -13.360, Z 91.800}
   LaserEnd_Ext()
   LIN {X 5.591, Y -13.360, Z 91.800}
   LaserStart_Ext()
   LIN {X 10.992, Y -13.360, Z 91.800}
   LaserEnd_Ext()
   LIN {X 11.015, Y -12.360, Z 91.800}
   LaserStart_Ext()
   LIN {X -3.759, Y -12.360, Z 91.800}
   LaserEnd_Ext()
   LIN {X -3.478, Y -11.360, Z 91.800}
   LaserStart_Ext()
   LIN {X 11.027, Y -11.360, Z 91.800}
   LaserEnd_Ext()
   LIN {X 11.039, Y -10.360, Z 91.800}
   LaserStart_Ext()
   LIN {X -3.196, Y -10.360, Z 91.800}
   LaserEnd_Ext()
   LIN {X -2.942, Y -9.360, Z 91.800}
   LaserStart_Ext()
   LIN {X 11.049, Y -9.360, Z 91.800}
   LaserEnd_Ext()
   LIN {X 11.025, Y -8.360, Z 91.800}
   LaserStart_Ext()
   LIN {X -2.704, Y -8.360, Z 91.800}
   LaserEnd_Ext()
   LIN {X -2.466, Y -7.360, Z 91.800}
   LaserStart_Ext()
   LIN {X 10.996, Y -7.360, Z 91.800}
   LaserEnd_Ext()
   LIN {X 10.969, Y -6.360, Z 91.800}
   LaserStart_Ext()
   LIN {X -2.261, Y -6.360, Z 91.800}
   LaserEnd_Ext()
   LIN {X -2.067, Y -5.360, Z 91.800}
   LaserStart_Ext()
   LIN {X 10.942, Y -5.360, Z 91.800}
   LaserEnd_Ext()
   LIN {X 10.910, Y -4.360, Z 91.800}
   LaserStart_Ext()
   LIN {X -1.874, Y -4.360, Z 91.800}
   LaserEnd_Ext()
   LIN {X -1.705, Y -3.360, Z 91.800}
   LaserStart_Ext()
   LIN {X 10.829, Y -3.360, Z 91.800}
   LaserEnd_Ext()
   LIN {X 10.748, Y -2.360, Z 91.800}
   LaserStart_Ext()
   LIN {X -1.553, Y -2.360, Z 91.800}
   LaserEnd_Ext()
   LIN {X -1.401, Y -1.360, Z 91.800}
   LaserStart_Ext()
   LIN {X 10.667, Y -1.360, Z 91.800}
   LaserEnd_Ext()
   LIN {X 10.586, Y -0.360, Z 91.800}
   LaserStart_Ext()
   LIN {X -1.280, Y -0.360, Z 91.800}
   LaserEnd_Ext()
   LIN {X -1.187, Y 0.640, Z 91.800}
   LaserStart_Ext()
   LIN {X 10.505, Y 0.640, Z 91.800}
   LaserEnd_Ext()
   LIN {X 10.424, Y 1.640, Z 91.800}
   LaserStart_Ext()
   LIN {X -1.094, Y 1.640, Z 91.800}
   LaserEnd_Ext()
   LIN {X -1.000, Y 2.640, Z 91.800}
   LaserStart_Ext()
   LIN {X 10.322, Y 2.640, Z 91.800}
   LaserEnd_Ext()
   LIN {X 10.166, Y 3.640, Z 91.800}
   LaserStart_Ext()
   LIN {X -0.907, Y 3.640, Z 91.800}
   LaserEnd_Ext()
   LIN {X -0.857, Y 4.640, Z 91.800}
   LaserStart_Ext()
   LIN {X 10.009, Y 4.640, Z 91.800}
   LaserEnd_Ext()
   LIN {X 9.852, Y 5.640, Z 91.800}
   LaserStart_Ext()
   LIN {X -0.844, Y 5.640, Z 91.800}
   LaserEnd_Ext()
   LIN {X -0.848, Y 6.640, Z 91.800}
   LaserStart_Ext()
   LIN {X 9.695, Y 6.640, Z 91.800}
   LaserEnd_Ext()
   LIN {X 9.538, Y 7.640, Z 91.800}
   LaserStart_Ext()
   LIN {X -0.851, Y 7.640, Z 91.800}
   LaserEnd_Ext()
   LIN {X -0.855, Y 8.640, Z 91.800}
   LaserStart_Ext()
   LIN {X 9.381, Y 8.640, Z 91.800}
   LaserEnd_Ext()
   LIN {X 9.224, Y 9.640, Z 91.800}
   LaserStart_Ext()
   LIN {X -0.859, Y 9.640, Z 91.800}
   LaserEnd_Ext()
   LIN {X -0.863, Y 10.640, Z 91.800}
   LaserStart_Ext()
   LIN {X 9.067, Y 10.640, Z 91.800}
   LaserEnd_Ext()
   LIN {X 8.910, Y 11.640, Z 91.800}
   LaserStart_Ext()
   LIN {X -0.867, Y 11.640, Z 91.800}
   LaserEnd_Ext()
   LIN {X -0.871, Y 12.640, Z 91.800}
   LaserStart_Ext()
   LIN {X 8.701, Y 12.640, Z 91.800}
   LaserEnd_Ext()
   LIN {X 8.446, Y 13.640, Z 91.800}
   LaserStart_Ext()
   LIN {X -0.937, Y 13.640, Z 91.800}
   LaserEnd_Ext()
   LIN {X -1.084, Y 14.640, Z 91.800}
   LaserStart_Ext()
   LIN {X 8.191, Y 14.640, Z 91.800}
   LaserEnd_Ext()
   LIN {X 7.936, Y 15.640, Z 91.800}
   LaserStart_Ext()
   LIN {X -1.251, Y 15.640, Z 91.800}
   LaserEnd_Ext()
   LIN {X -1.416, Y 16.640, Z 91.800}
   LaserStart_Ext()
   LIN {X 7.681, Y 16.640, Z 91.800}
   LaserEnd_Ext()
   LIN {X 7.426, Y 17.640, Z 91.800}
   LaserStart_Ext()
   LIN {X -1.560, Y 17.640, Z 91.800}
   LaserEnd_Ext()
   LIN {X -1.704, Y 18.640, Z 91.800}
   LaserStart_Ext()
   LIN {X 7.172, Y 18.640, Z 91.800}
   LaserEnd_Ext()
   LIN {X 6.917, Y 19.640, Z 91.800}
   LaserStart_Ext()
   LIN {X -1.849, Y 19.640, Z 91.800}
   LaserEnd_Ext()
   LIN {X -1.993, Y 20.640, Z 91.800}
   LaserStart_Ext()
   LIN {X 6.662, Y 20.640, Z 91.800}
   LaserEnd_Ext()
   LIN {X 6.409, Y 21.640, Z 91.800}
   LaserStart_Ext()
   LIN {X -2.138, Y 21.640, Z 91.800}
   LaserEnd_Ext()
   LIN {X -2.282, Y 22.640, Z 91.800}
   LaserStart_Ext()
   LIN {X 6.078, Y 22.640, Z 91.800}
   LaserEnd_Ext()
   LIN {X 5.729, Y 23.640, Z 91.800}
   LaserStart_Ext()
   LIN {X -2.426, Y 23.640, Z 91.800}
   LaserEnd_Ext()
   LIN {X -2.572, Y 24.640, Z 91.800}
   LaserStart_Ext()
   LIN {X 5.381, Y 24.640, Z 91.800}
   LaserEnd_Ext()
   LIN {X 5.032, Y 25.640, Z 91.800}
   LaserStart_Ext()
   LIN {X -2.795, Y 25.640, Z 91.800}
   LaserEnd_Ext()
   LIN {X -3.022, Y 26.640, Z 91.800}
   LaserStart_Ext()
   LIN {X 4.684, Y 26.640, Z 91.800}
   LaserEnd_Ext()
   LIN {X 4.335, Y 27.640, Z 91.800}
   LaserStart_Ext()
   LIN {X -3.283, Y 27.640, Z 91.800}
   LaserEnd_Ext()
   LIN {X -3.569, Y 28.640, Z 91.800}
   LaserStart_Ext()
   LIN {X 3.986, Y 28.640, Z 91.800}
   LaserEnd_Ext()
   LIN {X 3.638, Y 29.640, Z 91.800}
   LaserStart_Ext()
   LIN {X -3.856, Y 29.640, Z 91.800}
   LaserEnd_Ext()
   LIN {X -4.141, Y 30.640, Z 91.800}
   LaserStart_Ext()
   LIN {X 3.269, Y 30.640, Z 91.800}
   LaserEnd_Ext()
   LIN {X 2.859, Y 31.640, Z 91.800}
   LaserStart_Ext()
   LIN {X -4.482, Y 31.640, Z 91.800}
   LaserEnd_Ext()
   LIN {X -4.819, Y 32.640, Z 91.800}
   LaserStart_Ext()
   LIN {X 2.449, Y 32.640, Z 91.800}
   LaserEnd_Ext()
   LIN {X 2.030, Y 33.640, Z 91.800}
   LaserStart_Ext()
   LIN {X -5.156, Y 33.640, Z 91.800}
   LaserEnd_Ext()
   LIN {X -5.536, Y 34.640, Z 91.800}
   LaserStart_Ext()
   LIN {X 1.570, Y 34.640, Z 91.800}
   LaserEnd_Ext()
   LIN {X 1.109, Y 35.640, Z 91.800}
   LaserStart_Ext()
   LIN {X -5.921, Y 35.640, Z 91.800}
   LaserEnd_Ext()
   LIN {X -6.316, Y 36.640, Z 91.800}
   LaserStart_Ext()
   LIN {X 0.646, Y 36.640, Z 91.800}
   LaserEnd_Ext()
   LIN {X 0.183, Y 37.640, Z 91.800}
   LaserStart_Ext()
   LIN {X -6.741, Y 37.640, Z 91.800}
   LaserEnd_Ext()
   LIN {X -7.170, Y 38.640, Z 91.800}
   LaserStart_Ext()
   LIN {X -0.282, Y 38.640, Z 91.800}
   LaserEnd_Ext()
   LIN {X -0.787, Y 39.640, Z 91.800}
   LaserStart_Ext()
   LIN {X -7.627, Y 39.640, Z 91.800}
   LaserEnd_Ext()
   LIN {X -8.094, Y 40.640, Z 91.800}
   LaserStart_Ext()
   LIN {X -1.296, Y 40.640, Z 91.800}
   LaserEnd_Ext()
   LIN {X -1.821, Y 41.640, Z 91.800}
   LaserStart_Ext()
   LIN {X -8.483, Y 41.640, Z 91.800}
   LaserEnd_Ext()
   LIN {X -8.586, Y 42.640, Z 91.800}
   LaserStart_Ext()
   LIN {X -2.355, Y 42.640, Z 91.800}
   LaserEnd_Ext()
   LIN {X -2.904, Y 43.640, Z 91.800}
   LaserStart_Ext()
   LIN {X -8.349, Y 43.640, Z 91.800}
   LaserEnd_Ext()
   LIN {X -7.350, Y 44.640, Z 91.800}
   LaserStart_Ext()
   LIN {X -3.680, Y 44.640, Z 91.800}
   LaserEnd_Ext()
   LIN {X 0.347, Y -22.749, Z 92.650}
   LaserStart_Ext()
   LIN {X -0.316, Y -22.432, Z 92.650} C_DIS
   LIN {X -0.680, Y -22.008, Z 92.650} C_DIS
   LIN {X -1.669, Y -20.848, Z 92.650} C_DIS
   LIN {X -2.123, Y -19.262, Z 92.650} C_DIS
   LIN {X -2.245, Y -18.842, Z 92.650} C_DIS
   LIN {X -2.080, Y -18.100, Z 92.650} C_DIS
   LIN {X -1.616, Y -16.030, Z 92.650} C_DIS
   LIN {X -0.963, Y -15.282, Z 92.650} C_DIS
   LIN {X -0.219, Y -14.436, Z 92.650} C_DIS
   LIN {X 1.420, Y -13.706, Z 92.650} C_DIS
   LIN {X 1.782, Y -13.546, Z 92.650} C_DIS
   LIN {X 2.026, Y -13.552, Z 92.650} C_DIS
   LIN {X 3.939, Y -13.574, Z 92.650} C_DIS
   LIN {X 5.715, Y -14.435, Z 92.650} C_DIS
   LIN {X 5.852, Y -14.501, Z 92.650} C_DIS
   LIN {X 5.966, Y -14.650, Z 92.650} C_DIS
   LIN {X 7.387, Y -16.528, Z 92.650} C_DIS
   LIN {X 7.730, Y -18.604, Z 92.650} C_DIS
   LIN {X 7.747, Y -18.709, Z 92.650} C_DIS
   LIN {X 7.716, Y -18.811, Z 92.650} C_DIS
   LIN {X 7.140, Y -20.819, Z 92.650} C_DIS
   LIN {X 5.801, Y -22.341, Z 92.650} C_DIS
   LIN {X 5.637, Y -22.523, Z 92.650} C_DIS
   LIN {X 3.634, Y -23.372, Z 92.650} C_DIS
   LIN {X 2.534, Y -23.348, Z 92.650} C_DIS
   LIN {X 1.548, Y -23.325, Z 92.650} C_DIS
   LIN {X 0.347, Y -22.749, Z 92.650}
   LaserEnd_Ext()
   LIN {X -5.762, Y -15.540, Z 92.650}
   LaserStart_Ext()
   LIN {X -5.540, Y -14.852, Z 92.650} C_DIS
   LIN {X -4.836, Y -12.694, Z 92.650} C_DIS
   LIN {X -4.323, Y -10.873, Z 92.650} C_DIS
   LIN {X -3.969, Y -9.573, Z 92.650} C_DIS
   LIN {X -3.480, Y -7.518, Z 92.650} C_DIS
   LIN {X -3.030, Y -5.290, Z 92.650} C_DIS
   LIN {X -2.758, Y -3.879, Z 92.650} C_DIS
   LIN {X -2.427, Y -1.693, Z 92.650} C_DIS
   LIN {X -2.357, Y -1.236, Z 92.650} C_DIS
   LIN {X -2.255, Y -0.420, Z 92.650} C_DIS
   LIN {X -1.882, Y 3.582, Z 92.650} C_DIS
   LIN {X -1.814, Y 5.421, Z 92.650} C_DIS
   LIN {X -1.841, Y 12.536, Z 92.650} C_DIS
   LIN {X -2.005, Y 14.276, Z 92.650} C_DIS
   LIN {X -2.864, Y 19.427, Z 92.650} C_DIS
   LIN {X -3.650, Y 24.872, Z 92.650} C_DIS
   LIN {X -4.005, Y 26.445, Z 92.650} C_DIS
   LIN {X -4.540, Y 28.311, Z 92.650} C_DIS
   LIN {X -5.113, Y 30.333, Z 92.650} C_DIS
   LIN {X -5.565, Y 31.637, Z 92.650} C_DIS
   LIN {X -5.988, Y 32.892, Z 92.650} C_DIS
   LIN {X -6.170, Y 33.431, Z 92.650} C_DIS
   LIN {X -6.462, Y 34.190, Z 92.650} C_DIS
   LIN {X -7.163, Y 35.997, Z 92.650} C_DIS
   LIN {X -7.972, Y 37.887, Z 92.650} C_DIS
   LIN {X -8.095, Y 38.176, Z 92.650} C_DIS
   LIN {X -8.167, Y 38.333, Z 92.650} C_DIS
   LIN {X -8.764, Y 39.629, Z 92.650} C_DIS
   LIN {X -9.170, Y 40.484, Z 92.650} C_DIS
   LIN {X -9.301, Y 40.758, Z 92.650} C_DIS
   LIN {X -9.441, Y 41.239, Z 92.650} C_DIS
   LIN {X -9.700, Y 42.092, Z 92.650} C_DIS
   LIN {X -9.664, Y 42.751, Z 92.650} C_DIS
   LIN {X -9.624, Y 43.431, Z 92.650} C_DIS
   LIN {X -9.277, Y 44.202, Z 92.650} C_DIS
   LIN {X -8.960, Y 44.876, Z 92.650} C_DIS
   LIN {X -8.557, Y 45.282, Z 92.650} C_DIS
   LIN {X -7.243, Y 45.970, Z 92.650} C_DIS
   LIN {X -6.501, Y 46.437, Z 92.650} C_DIS
   LIN {X -5.521, Y 46.405, Z 92.650} C_DIS
   LIN {X -4.758, Y 46.381, Z 92.650} C_DIS
   LIN {X -4.272, Y 46.135, Z 92.650} C_DIS
   LIN {X -3.208, Y 45.592, Z 92.650} C_DIS
   LIN {X -2.357, Y 44.584, Z 92.650} C_DIS
   LIN {X -2.258, Y 44.468, Z 92.650} C_DIS
   LIN {X -2.198, Y 44.359, Z 92.650} C_DIS
   LIN {X -1.535, Y 43.155, Z 92.650} C_DIS
   LIN {X -0.910, Y 41.994, Z 92.650} C_DIS
   LIN {X -0.643, Y 41.493, Z 92.650} C_DIS
   LIN {X -0.004, Y 40.237, Z 92.650} C_DIS
   LIN {X 0.638, Y 38.981, Z 92.650} C_DIS
   LIN {X 1.232, Y 37.697, Z 92.650} C_DIS
   LIN {X 1.606, Y 36.894, Z 92.650} C_DIS
   LIN {X 3.173, Y 33.490, Z 92.650} C_DIS
   LIN {X 4.284, Y 30.779, Z 92.650} C_DIS
   LIN {X 6.976, Y 23.053, Z 92.650} C_DIS
   LIN {X 7.270, Y 22.267, Z 92.650} C_DIS
   LIN {X 7.402, Y 21.862, Z 92.650} C_DIS
   LIN {X 7.778, Y 20.378, Z 92.650} C_DIS
   LIN {X 9.857, Y 12.222, Z 92.650} C_DIS
   LIN {X 11.165, Y 3.884, Z 92.650} C_DIS
   LIN {X 11.421, Y 2.322, Z 92.650} C_DIS
   LIN {X 11.455, Y 1.969, Z 92.650} C_DIS
   LIN {X 11.502, Y 1.396, Z 92.650} C_DIS
   LIN {X 11.965, Y -4.326, Z 92.650} C_DIS
   LIN {X 11.975, Y -4.595, Z 92.650} C_DIS
   LIN {X 12.109, Y -9.110, Z 92.650} C_DIS
   LIN {X 12.101, Y -10.859, Z 92.650} C_DIS
   LIN {X 12.076, Y -12.914, Z 92.650} C_DIS
   LIN {X 11.959, Y -15.870, Z 92.650} C_DIS
   LIN {X -5.762, Y -15.540, Z 92.650}
   LaserEnd_Ext()
   LIN {X -5.762, Y -15.540, Z 92.650}
   LaserStart_Ext()
   LIN {X -5.865, Y -16.200, Z 92.650} C_DIS
   LIN {X -6.264, Y -18.670, Z 92.650} C_DIS
   LIN {X -5.548, Y -21.814, Z 92.650} C_DIS
   LIN {X -5.438, Y -22.287, Z 92.650} C_DIS
   LIN {X -5.239, Y -22.576, Z 92.650} C_DIS
   LIN {X -3.790, Y -24.707, Z 92.650} C_DIS
   LIN {X -1.538, Y -26.234, Z 92.650} C_DIS
   LIN {X -0.640, Y -26.833, Z 92.650} C_DIS
   LIN {X 0.433, Y -26.879, Z 92.650} C_DIS
   LIN {X 5.619, Y -26.974, Z 92.650} C_DIS
   LIN {X 8.249, Y -25.499, Z 92.650} C_DIS
   LIN {X 8.512, Y -25.347, Z 92.650} C_DIS
   LIN {X 8.635, Y -25.200, Z 92.650} C_DIS
   LIN {X 10.929, Y -22.169, Z 92.650} C_DIS
   LIN {X 11.319, Y -20.812, Z 92.650} C_DIS
   LIN {X 11.741, Y -19.126, Z 92.650} C_DIS
   LIN {X 11.959, Y -15.872, Z 92.650} C_DIS
   LIN {X -5.762, Y -15.540, Z 92.650}
   LaserEnd_Ext()
   LIN {X 10.602, Y 0.118, Z 92.650}
   LaserStart_Ext()
   LIN {X 10.602, Y -12.120, Z 92.650}
   LaserEnd_Ext()
   LIN {X 9.602, Y -22.265, Z 92.650}
   LaserStart_Ext()
   LIN {X 9.602, Y -19.709, Z 92.650}
   LaserEnd_Ext()
   LIN {X 9.602, Y -12.267, Z 92.650}
   LaserStart_Ext()
   LIN {X 9.602, Y 7.396, Z 92.650}
   LaserEnd_Ext()
   LIN {X 8.602, Y 13.097, Z 92.650}
   LaserStart_Ext()
   LIN {X 8.602, Y -12.414, Z 92.650}
   LaserEnd_Ext()
   LIN {X 8.602, Y -19.504, Z 92.650}
   LaserStart_Ext()
   LIN {X 8.602, Y -23.587, Z 92.650}
   LaserEnd_Ext()
   LIN {X 7.602, Y -24.715, Z 92.650}
   LaserStart_Ext()
   LIN {X 7.602, Y -19.299, Z 92.650}
   LaserEnd_Ext()
   LIN {X 7.602, Y -12.562, Z 92.650}
   LaserStart_Ext()
   LIN {X 7.602, Y 17.020, Z 92.650}
   LaserEnd_Ext()
   LIN {X 6.602, Y 20.949, Z 92.650}
   LaserStart_Ext()
   LIN {X 6.602, Y -12.709, Z 92.650}
   LaserEnd_Ext()
   LIN {X 6.602, Y -17.912, Z 92.650}
   LaserStart_Ext()
   LIN {X 6.602, Y -25.276, Z 92.650}
   LaserEnd_Ext()
   LIN {X 5.602, Y -25.837, Z 92.650}
   LaserStart_Ext()
   LIN {X 5.602, Y -15.826, Z 92.650}
   LaserEnd_Ext()
   LIN {X 5.602, Y -12.856, Z 92.650}
   LaserStart_Ext()
   LIN {X 5.602, Y 23.959, Z 92.650}
   LaserEnd_Ext()
   LIN {X 4.602, Y 26.827, Z 92.650}
   LaserStart_Ext()
   LIN {X 4.602, Y -13.005, Z 92.650}
   LaserEnd_Ext()
   LIN {X 4.602, Y -15.007, Z 92.650}
   LaserStart_Ext()
   LIN {X 4.602, Y -25.955, Z 92.650}
   LaserEnd_Ext()
   LIN {X 3.602, Y -25.937, Z 92.650}
   LaserStart_Ext()
   LIN {X 3.602, Y 29.696, Z 92.650}
   LaserEnd_Ext()
   LIN {X 2.602, Y 32.245, Z 92.650}
   LaserStart_Ext()
   LIN {X 2.602, Y -25.919, Z 92.650}
   LaserEnd_Ext()
   LIN {X 1.602, Y -25.900, Z 92.650}
   LaserStart_Ext()
   LIN {X 1.602, Y 34.510, Z 92.650}
   LaserEnd_Ext()
   LIN {X 0.602, Y 36.681, Z 92.650}
   LaserStart_Ext()
   LIN {X 0.602, Y -25.882, Z 92.650}
   LaserEnd_Ext()
   LIN {X -0.398, Y -25.792, Z 92.650}
   LaserStart_Ext()
   LIN {X -0.398, Y -16.155, Z 92.650}
   LaserEnd_Ext()
   LIN {X -0.398, Y -13.774, Z 92.650}
   LaserStart_Ext()
   LIN {X -0.398, Y 38.810, Z 92.650}
   LaserEnd_Ext()
   LIN {X -1.398, Y 40.772, Z 92.650}
   LaserStart_Ext()
   LIN {X -1.398, Y 16.716, Z 92.650}
   LaserEnd_Ext()
   LIN {X -1.398, Y -1.579, Z 92.650}
   LaserStart_Ext()
   LIN {X -1.398, Y -13.886, Z 92.650}
   LaserEnd_Ext()
   LIN {X -1.398, Y -17.328, Z 92.650}
   LaserStart_Ext()
   LIN {X -1.398, Y -25.120, Z 92.650}
   LaserEnd_Ext()
   LIN {X -2.398, Y -24.443, Z 92.650}
   LaserStart_Ext()
   LIN {X -2.398, Y -17.250, Z 92.650}
   LaserEnd_Ext()
   LIN {X -2.398, Y -14.034, Z 92.650}
   LaserStart_Ext()
   LIN {X -2.398, Y -7.214, Z 92.650}
   LaserEnd_Ext()
   LIN {X -2.398, Y 23.199, Z 92.650}
   LaserStart_Ext()
   LIN {X -2.398, Y 42.650, Z 92.650}
   LaserEnd_Ext()
   LIN {X -3.398, Y 44.267, Z 92.650}
   LaserStart_Ext()
   LIN {X -3.398, Y 27.956, Z 92.650}
   LaserEnd_Ext()
   LIN {X -3.398, Y -11.277, Z 92.650}
   LaserStart_Ext()
   LIN {X -3.398, Y -14.181, Z 92.650}
   LaserEnd_Ext()
   LIN {X -3.398, Y -17.045, Z 92.650}
   LaserStart_Ext()
   LIN {X -3.398, Y -23.505, Z 92.650}
   LaserEnd_Ext()
   LIN {X -4.398, Y -22.035, Z 92.650}
   LaserStart_Ext()
   LIN {X -4.398, Y -16.840, Z 92.650}
   LaserEnd_Ext()
   LIN {X -4.398, Y 31.323, Z 92.650}
   LaserStart_Ext()
   LIN {X -4.398, Y 45.077, Z 92.650}
   LaserEnd_Ext()
   LIN {X -5.398, Y 45.400, Z 92.650}
   LaserStart_Ext()
   LIN {X -5.398, Y 34.210, Z 92.650}
   LaserEnd_Ext()
   LIN {X -6.398, Y 36.752, Z 92.650}
   LaserStart_Ext()
   LIN {X -6.398, Y 45.320, Z 92.650}
   LaserEnd_Ext()
   LIN {X -7.398, Y 44.760, Z 92.650}
   LaserStart_Ext()
   LIN {X -7.398, Y 39.055, Z 92.650}
   LaserEnd_Ext()
   LIN {X -8.398, Y 41.235, Z 92.650}
   LaserStart_Ext()
   LIN {X -8.398, Y 43.718, Z 92.650}
   LaserEnd_Ext()
   LIN {X -0.225, Y -22.381, Z 93.500}
   LaserStart_Ext()
   LIN {X -1.458, Y -20.946, Z 93.500} C_DIS
   LIN {X -1.582, Y -20.801, Z 93.500} C_DIS
   LIN {X -1.639, Y -20.601, Z 93.500} C_DIS
   LIN {X -2.162, Y -18.797, Z 93.500} C_DIS
   LIN {X -1.598, Y -16.254, Z 93.500} C_DIS
   LIN {X -1.534, Y -15.973, Z 93.500} C_DIS
   LIN {X -1.334, Y -15.748, Z 93.500} C_DIS
   LIN {X -0.111, Y -14.359, Z 93.500} C_DIS
   LIN {X 0.958, Y -13.883, Z 93.500} C_DIS
   LIN {X 1.843, Y -13.492, Z 93.500} C_DIS
   LIN {X 3.200, Y -13.504, Z 93.500} C_DIS
   LIN {X 4.009, Y -13.514, Z 93.500} C_DIS
   LIN {X 4.585, Y -13.793, Z 93.500} C_DIS
   LIN {X 5.924, Y -14.435, Z 93.500} C_DIS
   LIN {X 7.038, Y -15.897, Z 93.500} C_DIS
   LIN {X 7.464, Y -16.459, Z 93.500} C_DIS
   LIN {X 7.578, Y -17.150, Z 93.500} C_DIS
   LIN {X 7.829, Y -18.639, Z 93.500} C_DIS
   LIN {X 7.532, Y -19.737, Z 93.500} C_DIS
   LIN {X 7.256, Y -20.698, Z 93.500} C_DIS
   LIN {X 6.514, Y -21.541, Z 93.500} C_DIS
   LIN {X 5.716, Y -22.467, Z 93.500} C_DIS
   LIN {X 3.719, Y -23.313, Z 93.500} C_DIS
   LIN {X 2.071, Y -23.279, Z 93.500} C_DIS
   LIN {X 1.640, Y -23.270, Z 93.500} C_DIS
   LIN {X 1.368, Y -23.142, Z 93.500} C_DIS
   LIN {X -0.225, Y -22.381, Z 93.500}
   LaserEnd_Ext()
   LIN {X -8.767, Y 39.548, Z 93.500}
   LaserStart_Ext()
   LIN {X -8.819, Y 39.659, Z 93.500} C_DIS
   LIN {X -8.883, Y 39.794, Z 93.500} C_DIS
   LIN {X -9.358, Y 40.788, Z 93.500} C_DIS
   LIN {X -9.602, Y 41.621, Z 93.500} C_DIS
   LIN {X -9.765, Y 42.158, Z 93.500} C_DIS
   LIN {X -9.748, Y 42.637, Z 93.500} C_DIS
   LIN {X -9.703, Y 43.392, Z 93.500} C_DIS
   LIN {X -9.265, Y 44.365, Z 93.500} C_DIS
   LIN {X -9.014, Y 44.925, Z 93.500} C_DIS
   LIN {X -8.582, Y 45.354, Z 93.500} C_DIS
   LIN {X -8.263, Y 45.676, Z 93.500} C_DIS
   LIN {X -7.481, Y 46.084, Z 93.500} C_DIS
   LIN {X -6.573, Y 46.472, Z 93.500} C_DIS
   LIN {X -5.850, Y 46.452, Z 93.500} C_DIS
   LIN {X -4.829, Y 46.421, Z 93.500} C_DIS
   LIN {X -3.587, Y 45.791, Z 93.500} C_DIS
   LIN {X -3.277, Y 45.635, Z 93.500} C_DIS
   LIN {X -3.116, Y 45.447, Z 93.500} C_DIS
   LIN {X -2.324, Y 44.513, Z 93.500} C_DIS
   LIN {X -1.626, Y 43.253, Z 93.500} C_DIS
   LIN {X -1.515, Y 43.049, Z 93.500} C_DIS
   LIN {X -0.699, Y 41.535, Z 93.500} C_DIS
   LIN {X -0.033, Y 40.239, Z 93.500} C_DIS
   LIN {X 0.634, Y 38.932, Z 93.500} C_DIS
   LIN {X 0.870, Y 38.423, Z 93.500} C_DIS
   LIN {X 1.340, Y 37.412, Z 93.500} C_DIS
   LIN {X 3.310, Y 33.132, Z 93.500} C_DIS
   LIN {X 4.226, Y 30.896, Z 93.500} C_DIS
   LIN {X 6.447, Y 24.526, Z 93.500} C_DIS
   LIN {X 7.161, Y 22.609, Z 93.500} C_DIS
   LIN {X 7.485, Y 21.624, Z 93.500} C_DIS
   LIN {X 8.400, Y 18.007, Z 93.500} C_DIS
   LIN {X 9.896, Y 12.136, Z 93.500} C_DIS
   LIN {X 10.838, Y 6.134, Z 93.500} C_DIS
   LIN {X 11.471, Y 2.262, Z 93.500} C_DIS
   LIN {X 11.557, Y 1.387, Z 93.500} C_DIS
   LIN {X 11.672, Y -0.033, Z 93.500} C_DIS
   LIN {X 12.013, Y -4.247, Z 93.500} C_DIS
   LIN {X 12.083, Y -6.163, Z 93.500} C_DIS
   LIN {X 12.169, Y -9.030, Z 93.500} C_DIS
   LIN {X 12.154, Y -12.068, Z 93.500} C_DIS
   LIN {X 12.144, Y -12.834, Z 93.500} C_DIS
   LIN {X 12.101, Y -13.937, Z 93.500} C_DIS
   LIN {X 12.035, Y -15.792, Z 93.500} C_DIS
   LIN {X 11.961, Y -17.004, Z 93.500} C_DIS
   LIN {X 11.824, Y -19.047, Z 93.500} C_DIS
   LIN {X 11.108, Y -21.908, Z 93.500} C_DIS
   LIN {X 8.637, Y -25.251, Z 93.500} C_DIS
   LIN {X 7.704, Y -25.763, Z 93.500} C_DIS
   LIN {X 5.569, Y -26.960, Z 93.500} C_DIS
   LIN {X 2.048, Y -26.896, Z 93.500} C_DIS
   LIN {X -0.535, Y -26.784, Z 93.500} C_DIS
   LIN {X -2.698, Y -25.342, Z 93.500} C_DIS
   LIN {X -3.690, Y -24.669, Z 93.500} C_DIS
   LIN {X -4.328, Y -23.731, Z 93.500} C_DIS
   LIN {X -5.347, Y -22.249, Z 93.500} C_DIS
   LIN {X -5.911, Y -19.823, Z 93.500} C_DIS
   LIN {X -6.182, Y -18.634, Z 93.500} C_DIS
   LIN {X -6.031, Y -17.700, Z 93.500} C_DIS
   LIN {X -5.687, Y -15.502, Z 93.500} C_DIS
   LIN {X -4.951, Y -13.216, Z 93.500} C_DIS
   LIN {X -4.775, Y -12.677, Z 93.500} C_DIS
   LIN {X -4.647, Y -12.223, Z 93.500} C_DIS
   LIN {X -3.860, Y -9.331, Z 93.500} C_DIS
   LIN {X -3.536, Y -7.973, Z 93.500} C_DIS
   LIN {X -2.848, Y -4.558, Z 93.500} C_DIS
   LIN {X -2.742, Y -4.009, Z 93.500} C_DIS
   LIN {X -2.476, Y -2.256, Z 93.500} C_DIS
   LIN {X -2.341, Y -1.367, Z 93.500} C_DIS
   LIN {X -2.215, Y -0.357, Z 93.500} C_DIS
   LIN {X -1.881, Y 3.223, Z 93.500} C_DIS
   LIN {X -1.787, Y 5.772, Z 93.500} C_DIS
   LIN {X -1.811, Y 12.176, Z 93.500} C_DIS
   LIN {X -2.055, Y 14.772, Z 93.500} C_DIS
   LIN {X -3.336, Y 22.455, Z 93.500} C_DIS
   LIN {X -3.743, Y 25.271, Z 93.500} C_DIS
   LIN {X -3.927, Y 26.084, Z 93.500} C_DIS
   LIN {X -4.203, Y 27.049, Z 93.500} C_DIS
   LIN {X -5.135, Y 30.336, Z 93.500} C_DIS
   LIN {X -5.870, Y 32.458, Z 93.500} C_DIS
   LIN {X -6.210, Y 33.467, Z 93.500} C_DIS
   LIN {X -7.049, Y 35.618, Z 93.500} C_DIS
   LIN {X -7.210, Y 36.031, Z 93.500} C_DIS
   LIN {X -7.327, Y 36.305, Z 93.500} C_DIS
   LIN {X -8.147, Y 38.208, Z 93.500} C_DIS
   LIN {X -8.767, Y 39.548, Z 93.500}
   LaserEnd_Ext()
   LIN {X -3.643, Y 44.522, Z 93.500}
   LaserStart_Ext()
   LIN {X -8.001, Y 44.522, Z 93.500}
   LaserEnd_Ext()
   LIN {X -8.548, Y 43.522, Z 93.500}
   LaserStart_Ext()
   LIN {X -2.918, Y 43.522, Z 93.500}
   LaserEnd_Ext()
   LIN {X -2.367, Y 42.522, Z 93.500}
   LaserStart_Ext()
   LIN {X -8.751, Y 42.522, Z 93.500}
   LaserEnd_Ext()
   LIN {X -8.531, Y 41.522, Z 93.500}
   LaserStart_Ext()
   LIN {X -1.828, Y 41.522, Z 93.500}
   LaserEnd_Ext()
   LIN {X -1.303, Y 40.522, Z 93.500}
   LaserStart_Ext()
   LIN {X -8.123, Y 40.522, Z 93.500}
   LaserEnd_Ext()
   LIN {X -7.653, Y 39.522, Z 93.500}
   LaserStart_Ext()
   LIN {X -0.790, Y 39.522, Z 93.500}
   LaserEnd_Ext()
   LIN {X -0.279, Y 38.522, Z 93.500}
   LaserStart_Ext()
   LIN {X -7.193, Y 38.522, Z 93.500}
   LaserEnd_Ext()
   LIN {X -6.762, Y 37.522, Z 93.500}
   LaserStart_Ext()
   LIN {X 0.186, Y 37.522, Z 93.500}
   LaserEnd_Ext()
   LIN {X 0.649, Y 36.522, Z 93.500}
   LaserStart_Ext()
   LIN {X -6.332, Y 36.522, Z 93.500}
   LaserEnd_Ext()
   LIN {X -5.938, Y 35.522, Z 93.500}
   LaserStart_Ext()
   LIN {X 1.109, Y 35.522, Z 93.500}
   LaserEnd_Ext()
   LIN {X 1.569, Y 34.522, Z 93.500}
   LaserStart_Ext()
   LIN {X -5.548, Y 34.522, Z 93.500}
   LaserEnd_Ext()
   LIN {X -5.174, Y 33.522, Z 93.500}
   LaserStart_Ext()
   LIN {X 2.030, Y 33.522, Z 93.500}
   LaserEnd_Ext()
   LIN {X 2.479, Y 32.522, Z 93.500}
   LaserStart_Ext()
   LIN {X -4.834, Y 32.522, Z 93.500}
   LaserEnd_Ext()
   LIN {X -4.488, Y 31.522, Z 93.500}
   LaserStart_Ext()
   LIN {X 2.889, Y 31.522, Z 93.500}
   LaserEnd_Ext()
   LIN {X 3.298, Y 30.522, Z 93.500}
   LaserStart_Ext()
   LIN {X -4.148, Y 30.522, Z 93.500}
   LaserEnd_Ext()
   LIN {X -3.865, Y 29.522, Z 93.500}
   LaserStart_Ext()
   LIN {X 3.646, Y 29.522, Z 93.500}
   LaserEnd_Ext()
   LIN {X 3.995, Y 28.522, Z 93.500}
   LaserStart_Ext()
   LIN {X -3.581, Y 28.522, Z 93.500}
   LaserEnd_Ext()
   LIN {X -3.298, Y 27.522, Z 93.500}
   LaserStart_Ext()
   LIN {X 4.343, Y 27.522, Z 93.500}
   LaserEnd_Ext()
   LIN {X 4.692, Y 26.522, Z 93.500}
   LaserStart_Ext()
   LIN {X -3.012, Y 26.522, Z 93.500}
   LaserEnd_Ext()
   LIN {X -2.774, Y 25.522, Z 93.500}
   LaserStart_Ext()
   LIN {X 5.041, Y 25.522, Z 93.500}
   LaserEnd_Ext()
   LIN {X 5.389, Y 24.522, Z 93.500}
   LaserStart_Ext()
   LIN {X -2.624, Y 24.522, Z 93.500}
   LaserEnd_Ext()
   LIN {X -2.480, Y 23.522, Z 93.500}
   LaserStart_Ext()
   LIN {X 5.754, Y 23.522, Z 93.500}
   LaserEnd_Ext()
   LIN {X 6.127, Y 22.522, Z 93.500}
   LaserStart_Ext()
   LIN {X -2.334, Y 22.522, Z 93.500}
   LaserEnd_Ext()
   LIN {X -2.167, Y 21.522, Z 93.500}
   LaserStart_Ext()
   LIN {X 6.466, Y 21.522, Z 93.500}
   LaserEnd_Ext()
   LIN {X 6.732, Y 20.522, Z 93.500}
   LaserStart_Ext()
   LIN {X -2.000, Y 20.522, Z 93.500}
   LaserEnd_Ext()
   LIN {X -1.833, Y 19.522, Z 93.500}
   LaserStart_Ext()
   LIN {X 6.985, Y 19.522, Z 93.500}
   LaserEnd_Ext()
   LIN {X 7.238, Y 18.522, Z 93.500}
   LaserStart_Ext()
   LIN {X -1.667, Y 18.522, Z 93.500}
   LaserEnd_Ext()
   LIN {X -1.500, Y 17.522, Z 93.500}
   LaserStart_Ext()
   LIN {X 7.492, Y 17.522, Z 93.500}
   LaserEnd_Ext()
   LIN {X 7.747, Y 16.522, Z 93.500}
   LaserStart_Ext()
   LIN {X -1.333, Y 16.522, Z 93.500}
   LaserEnd_Ext()
   LIN {X -1.167, Y 15.522, Z 93.500}
   LaserStart_Ext()
   LIN {X 8.001, Y 15.522, Z 93.500}
   LaserEnd_Ext()
   LIN {X 8.256, Y 14.522, Z 93.500}
   LaserStart_Ext()
   LIN {X -1.027, Y 14.522, Z 93.500}
   LaserEnd_Ext()
   LIN {X -0.933, Y 13.522, Z 93.500}
   LaserStart_Ext()
   LIN {X 8.511, Y 13.522, Z 93.500}
   LaserEnd_Ext()
   LIN {X 8.766, Y 12.522, Z 93.500}
   LaserStart_Ext()
   LIN {X -0.839, Y 12.522, Z 93.500}
   LaserEnd_Ext()
   LIN {X -0.809, Y 11.522, Z 93.500}
   LaserStart_Ext()
   LIN {X 8.980, Y 11.522, Z 93.500}
   LaserEnd_Ext()
   LIN {X 9.137, Y 10.522, Z 93.500}
   LaserStart_Ext()
   LIN {X -0.805, Y 10.522, Z 93.500}
   LaserEnd_Ext()
   LIN {X -0.801, Y 9.522, Z 93.500}
   LaserStart_Ext()
   LIN {X 9.294, Y 9.522, Z 93.500}
   LaserEnd_Ext()
   LIN {X 9.451, Y 8.522, Z 93.500}
   LaserStart_Ext()
   LIN {X -0.797, Y 8.522, Z 93.500}
   LaserEnd_Ext()
   LIN {X -0.793, Y 7.522, Z 93.500}
   LaserStart_Ext()
   LIN {X 9.608, Y 7.522, Z 93.500}
   LaserEnd_Ext()
   LIN {X 9.765, Y 6.522, Z 93.500}
   LaserStart_Ext()
   LIN {X -0.790, Y 6.522, Z 93.500}
   LaserEnd_Ext()
   LIN {X -0.795, Y 5.522, Z 93.500}
   LaserStart_Ext()
   LIN {X 9.925, Y 5.522, Z 93.500}
   LaserEnd_Ext()
   LIN {X 10.088, Y 4.522, Z 93.500}
   LaserStart_Ext()
   LIN {X -0.832, Y 4.522, Z 93.500}
   LaserEnd_Ext()
   LIN {X -0.869, Y 3.522, Z 93.500}
   LaserStart_Ext()
   LIN {X 10.252, Y 3.522, Z 93.500}
   LaserEnd_Ext()
   LIN {X 10.415, Y 2.522, Z 93.500}
   LaserStart_Ext()
   LIN {X -0.942, Y 2.522, Z 93.500}
   LaserEnd_Ext()
   LIN {X -1.035, Y 1.522, Z 93.500}
   LaserStart_Ext()
   LIN {X 10.539, Y 1.522, Z 93.500}
   LaserEnd_Ext()
   LIN {X 10.624, Y 0.522, Z 93.500}
   LaserStart_Ext()
   LIN {X -1.129, Y 0.522, Z 93.500}
   LaserEnd_Ext()
   LIN {X -1.222, Y -0.478, Z 93.500}
   LaserStart_Ext()
   LIN {X 10.705, Y -0.478, Z 93.500}
   LaserEnd_Ext()
   LIN {X 10.786, Y -1.478, Z 93.500}
   LaserStart_Ext()
   LIN {X -1.347, Y -1.478, Z 93.500}
   LaserEnd_Ext()
   LIN {X -1.498, Y -2.478, Z 93.500}
   LaserStart_Ext()
   LIN {X 10.867, Y -2.478, Z 93.500}
   LaserEnd_Ext()
   LIN {X 10.948, Y -3.478, Z 93.500}
   LaserStart_Ext()
   LIN {X -1.650, Y -3.478, Z 93.500}
   LaserEnd_Ext()
   LIN {X -1.814, Y -4.478, Z 93.500}
   LaserStart_Ext()
   LIN {X 11.021, Y -4.478, Z 93.500}
   LaserEnd_Ext()
   LIN {X 11.058, Y -5.478, Z 93.500}
   LaserStart_Ext()
   LIN {X -2.013, Y -5.478, Z 93.500}
   LaserEnd_Ext()
   LIN {X -2.215, Y -6.478, Z 93.500}
   LaserStart_Ext()
   LIN {X 11.092, Y -6.478, Z 93.500}
   LaserEnd_Ext()
   LIN {X 11.122, Y -7.478, Z 93.500}
   LaserStart_Ext()
   LIN {X -2.416, Y -7.478, Z 93.500}
   LaserEnd_Ext()
   LIN {X -2.628, Y -8.478, Z 93.500}
   LaserStart_Ext()
   LIN {X 11.152, Y -8.478, Z 93.500}
   LaserEnd_Ext()
   LIN {X 11.166, Y -9.478, Z 93.500}
   LaserStart_Ext()
   LIN {X -2.867, Y -9.478, Z 93.500}
   LaserEnd_Ext()
   LIN {X -3.136, Y -10.478, Z 93.500}
   LaserStart_Ext()
   LIN {X 11.162, Y -10.478, Z 93.500}
   LaserEnd_Ext()
   LIN {X 11.157, Y -11.478, Z 93.500}
   LaserStart_Ext()
   LIN {X -3.408, Y -11.478, Z 93.500}
   LaserEnd_Ext()
   LIN {X -3.680, Y -12.478, Z 93.500}
   LaserStart_Ext()
   LIN {X 11.149, Y -12.478, Z 93.500}
   LaserEnd_Ext()
   LIN {X 11.118, Y -13.478, Z 93.500}
   LaserStart_Ext()
   LIN {X 6.241, Y -13.478, Z 93.500}
   LaserEnd_Ext()
   LIN {X -0.582, Y -13.478, Z 93.500}
   LaserStart_Ext()
   LIN {X -3.985, Y -13.478, Z 93.500}
   LaserEnd_Ext()
   LIN {X -4.307, Y -14.478, Z 93.500}
   LaserStart_Ext()
   LIN {X -1.548, Y -14.478, Z 93.500}
   LaserEnd_Ext()
   LIN {X 7.214, Y -14.478, Z 93.500}
   LaserStart_Ext()
   LIN {X 11.081, Y -14.478, Z 93.500}
   LaserEnd_Ext()
   LIN {X 11.045, Y -15.478, Z 93.500}
   LaserStart_Ext()
   LIN {X 7.975, Y -15.478, Z 93.500}
   LaserEnd_Ext()
   LIN {X -2.403, Y -15.478, Z 93.500}
   LaserStart_Ext()
   LIN {X -4.629, Y -15.478, Z 93.500}
   LaserEnd_Ext()
   LIN {X -4.828, Y -16.478, Z 93.500}
   LaserStart_Ext()
   LIN {X -2.672, Y -16.478, Z 93.500}
   LaserEnd_Ext()
   LIN {X 8.480, Y -16.478, Z 93.500}
   LaserStart_Ext()
   LIN {X 10.991, Y -16.478, Z 93.500}
   LaserEnd_Ext()
   LIN {X 10.927, Y -17.478, Z 93.500}
   LaserStart_Ext()
   LIN {X 8.647, Y -17.478, Z 93.500}
   LaserEnd_Ext()
   LIN {X -2.894, Y -17.478, Z 93.500}
   LaserStart_Ext()
   LIN {X -4.985, Y -17.478, Z 93.500}
   LaserEnd_Ext()
   LIN {X -5.144, Y -18.478, Z 93.500}
   LaserStart_Ext()
   LIN {X -3.116, Y -18.478, Z 93.500}
   LaserEnd_Ext()
   LIN {X 8.816, Y -18.478, Z 93.500}
   LaserStart_Ext()
   LIN {X 10.860, Y -18.478, Z 93.500}
   LaserEnd_Ext()
   LIN {X 10.685, Y -19.478, Z 93.500}
   LaserStart_Ext()
   LIN {X 8.638, Y -19.478, Z 93.500}
   LaserEnd_Ext()
   LIN {X -3.006, Y -19.478, Z 93.500}
   LaserStart_Ext()
   LIN {X -4.964, Y -19.478, Z 93.500}
   LaserEnd_Ext()
   LIN {X -4.732, Y -20.478, Z 93.500}
   LaserStart_Ext()
   LIN {X -2.716, Y -20.478, Z 93.500}
   LaserEnd_Ext()
   LIN {X 8.359, Y -20.478, Z 93.500}
   LaserStart_Ext()
   LIN {X 10.435, Y -20.478, Z 93.500}
   LaserEnd_Ext()
   LIN {X 10.185, Y -21.478, Z 93.500}
   LaserStart_Ext()
   LIN {X 7.901, Y -21.478, Z 93.500}
   LaserEnd_Ext()
   LIN {X -2.318, Y -21.478, Z 93.500}
   LaserStart_Ext()
   LIN {X -4.500, Y -21.478, Z 93.500}
   LaserEnd_Ext()
   LIN {X -3.976, Y -22.478, Z 93.500}
   LaserStart_Ext()
   LIN {X -1.460, Y -22.478, Z 93.500}
   LaserEnd_Ext()
   LIN {X 7.027, Y -22.478, Z 93.500}
   LaserStart_Ext()
   LIN {X 9.447, Y -22.478, Z 93.500}
   LaserEnd_Ext()
   LIN {X 8.706, Y -23.478, Z 93.500}
   LaserStart_Ext()
   LIN {X 5.893, Y -23.478, Z 93.500}
   LaserEnd_Ext()
   LIN {X -0.249, Y -23.478, Z 93.500}
   LaserStart_Ext()
   LIN {X -3.290, Y -23.478, Z 93.500}
   LaserEnd_Ext()
   LIN {X -2.189, Y -24.478, Z 93.500}
   LaserStart_Ext()
   LIN {X 7.965, Y -24.478, Z 93.500}
   LaserEnd_Ext()
   LIN {X 6.167, Y -25.478, Z 93.500}
   LaserStart_Ext()
   LIN {X -0.691, Y -25.478, Z 93.500}
   LaserEnd_Ext()
   LIN {X 6.917, Y -15.578, Z 94.350}
   LaserStart_Ext()
   LIN {X 7.541, Y -16.391, Z 94.350} C_DIS
   LIN {X 7.674, Y -17.165, Z 94.350} C_DIS
   LIN {X 7.911, Y -18.569, Z 94.350} C_DIS
   LIN {X 7.462, Y -20.228, Z 94.350} C_DIS
   LIN {X 7.353, Y -20.611, Z 94.350} C_DIS
   LIN {X 7.080, Y -20.919, Z 94.350} C_DIS
   LIN {X 5.793, Y -22.413, Z 94.350} C_DIS
   LIN {X 3.804, Y -23.255, Z 94.350} C_DIS
   LIN {X 1.734, Y -23.215, Z 94.350} C_DIS
   LIN {X 0.335, Y -22.555, Z 94.350} C_DIS
   LIN {X -0.135, Y -22.331, Z 94.350} C_DIS
   LIN {X -0.579, Y -21.813, Z 94.350} C_DIS
   LIN {X -1.495, Y -20.753, Z 94.350} C_DIS
   LIN {X -1.893, Y -19.395, Z 94.350} C_DIS
   LIN {X -2.080, Y -18.751, Z 94.350} C_DIS
   LIN {X -1.917, Y -18.017, Z 94.350} C_DIS
   LIN {X -1.436, Y -15.886, Z 94.350} C_DIS
   LIN {X -0.053, Y -14.337, Z 94.350} C_DIS
   LIN {X 0.092, Y -14.240, Z 94.350} C_DIS
   LIN {X 1.913, Y -13.437, Z 94.350} C_DIS
   LIN {X 3.409, Y -13.450, Z 94.350} C_DIS
   LIN {X 4.079, Y -13.453, Z 94.350} C_DIS
   LIN {X 4.809, Y -13.801, Z 94.350} C_DIS
   LIN {X 5.997, Y -14.370, Z 94.350} C_DIS
   LIN {X 6.917, Y -15.578, Z 94.350}
   LaserEnd_Ext()
   LIN {X -1.660, Y 43.247, Z 94.350}
   LaserStart_Ext()
   LIN {X -0.974, Y 41.983, Z 94.350} C_DIS
   LIN {X -0.750, Y 41.569, Z 94.350} C_DIS
   LIN {X -0.097, Y 40.297, Z 94.350} C_DIS
   LIN {X 0.631, Y 38.883, Z 94.350} C_DIS
   LIN {X 1.074, Y 37.931, Z 94.350} C_DIS
   LIN {X 3.448, Y 32.774, Z 94.350} C_DIS
   LIN {X 4.169, Y 31.014, Z 94.350} C_DIS
   LIN {X 5.917, Y 25.998, Z 94.350} C_DIS
   LIN {X 7.053, Y 22.951, Z 94.350} C_DIS
   LIN {X 7.567, Y 21.386, Z 94.350} C_DIS
   LIN {X 9.022, Y 15.636, Z 94.350} C_DIS
   LIN {X 9.936, Y 12.049, Z 94.350} C_DIS
   LIN {X 10.511, Y 8.383, Z 94.350} C_DIS
   LIN {X 11.521, Y 2.203, Z 94.350} C_DIS
   LIN {X 11.659, Y 0.805, Z 94.350} C_DIS
   LIN {X 11.842, Y -1.461, Z 94.350} C_DIS
   LIN {X 12.061, Y -4.167, Z 94.350} C_DIS
   LIN {X 12.192, Y -7.731, Z 94.350} C_DIS
   LIN {X 12.228, Y -8.951, Z 94.350} C_DIS
   LIN {X 12.216, Y -11.410, Z 94.350} C_DIS
   LIN {X 12.213, Y -12.755, Z 94.350} C_DIS
   LIN {X 12.197, Y -13.262, Z 94.350} C_DIS
   LIN {X 12.110, Y -15.712, Z 94.350} C_DIS
   LIN {X 11.963, Y -18.136, Z 94.350} C_DIS
   LIN {X 11.907, Y -18.968, Z 94.350} C_DIS
   LIN {X 11.616, Y -20.133, Z 94.350} C_DIS
   LIN {X 11.195, Y -21.843, Z 94.350} C_DIS
   LIN {X 10.378, Y -22.977, Z 94.350} C_DIS
   LIN {X 8.767, Y -25.152, Z 94.350} C_DIS
   LIN {X 6.646, Y -26.315, Z 94.350} C_DIS
   LIN {X 5.520, Y -26.946, Z 94.350} C_DIS
   LIN {X 3.663, Y -26.912, Z 94.350} C_DIS
   LIN {X -0.430, Y -26.736, Z 94.350} C_DIS
   LIN {X -3.193, Y -24.893, Z 94.350} C_DIS
   LIN {X -3.590, Y -24.631, Z 94.350} C_DIS
   LIN {X -3.759, Y -24.388, Z 94.350} C_DIS
   LIN {X -5.257, Y -22.210, Z 94.350} C_DIS
   LIN {X -5.954, Y -19.213, Z 94.350} C_DIS
   LIN {X -6.100, Y -18.598, Z 94.350} C_DIS
   LIN {X -6.006, Y -17.975, Z 94.350} C_DIS
   LIN {X -5.613, Y -15.464, Z 94.350} C_DIS
   LIN {X -4.975, Y -13.484, Z 94.350} C_DIS
   LIN {X -4.705, Y -12.631, Z 94.350} C_DIS
   LIN {X -4.296, Y -11.095, Z 94.350} C_DIS
   LIN {X -3.750, Y -9.089, Z 94.350} C_DIS
   LIN {X -3.593, Y -8.429, Z 94.350} C_DIS
   LIN {X -2.985, Y -5.416, Z 94.350} C_DIS
   LIN {X -2.772, Y -4.389, Z 94.350} C_DIS
   LIN {X -2.687, Y -3.895, Z 94.350} C_DIS
   LIN {X -2.322, Y -1.498, Z 94.350} C_DIS
   LIN {X -2.275, Y -1.098, Z 94.350} C_DIS
   LIN {X -2.174, Y -0.293, Z 94.350} C_DIS
   LIN {X -1.880, Y 2.864, Z 94.350} C_DIS
   LIN {X -1.759, Y 6.122, Z 94.350} C_DIS
   LIN {X -1.781, Y 11.816, Z 94.350} C_DIS
   LIN {X -2.106, Y 15.268, Z 94.350} C_DIS
   LIN {X -3.809, Y 25.484, Z 94.350} C_DIS
   LIN {X -3.836, Y 25.670, Z 94.350} C_DIS
   LIN {X -3.866, Y 25.787, Z 94.350} C_DIS
   LIN {X -5.157, Y 30.340, Z 94.350} C_DIS
   LIN {X -6.175, Y 33.278, Z 94.350} C_DIS
   LIN {X -6.251, Y 33.503, Z 94.350} C_DIS
   LIN {X -6.498, Y 34.135, Z 94.350} C_DIS
   LIN {X -7.256, Y 36.064, Z 94.350} C_DIS
   LIN {X -8.130, Y 38.080, Z 94.350} C_DIS
   LIN {X -8.198, Y 38.239, Z 94.350} C_DIS
   LIN {X -8.874, Y 39.689, Z 94.350} C_DIS
   LIN {X -9.258, Y 40.492, Z 94.350} C_DIS
   LIN {X -9.414, Y 40.817, Z 94.350} C_DIS
   LIN {X -9.543, Y 41.219, Z 94.350} C_DIS
   LIN {X -9.819, Y 42.124, Z 94.350} C_DIS
   LIN {X -9.787, Y 42.996, Z 94.350} C_DIS
   LIN {X -9.772, Y 43.396, Z 94.350} C_DIS
   LIN {X -9.508, Y 43.965, Z 94.350} C_DIS
   LIN {X -9.038, Y 45.013, Z 94.350} C_DIS
   LIN {X -8.628, Y 45.420, Z 94.350} C_DIS
   LIN {X -7.342, Y 46.210, Z 94.350} C_DIS
   LIN {X -6.644, Y 46.508, Z 94.350} C_DIS
   LIN {X -5.488, Y 46.475, Z 94.350} C_DIS
   LIN {X -4.900, Y 46.460, Z 94.350} C_DIS
   LIN {X -4.558, Y 46.289, Z 94.350} C_DIS
   LIN {X -3.346, Y 45.678, Z 94.350} C_DIS
   LIN {X -2.477, Y 44.661, Z 94.350} C_DIS
   LIN {X -2.390, Y 44.559, Z 94.350} C_DIS
   LIN {X -2.334, Y 44.459, Z 94.350} C_DIS
   LIN {X -1.660, Y 43.247, Z 94.350}
   LaserEnd_Ext()
   LIN {X -8.280, Y 44.259, Z 94.350}
   LaserStart_Ext()
   LIN {X -8.280, Y 40.764, Z 94.350}
   LaserEnd_Ext()
   LIN {X -7.280, Y 38.634, Z 94.350}
   LaserStart_Ext()
   LIN {X -7.280, Y 45.074, Z 94.350}
   LaserEnd_Ext()
   LIN {X -6.280, Y 45.497, Z 94.350}
   LaserStart_Ext()
   LIN {X -6.280, Y 36.315, Z 94.350}
   LaserEnd_Ext()
   LIN {X -5.280, Y 33.752, Z 94.350}
   LaserStart_Ext()
   LIN {X -5.280, Y 45.470, Z 94.350}
   LaserEnd_Ext()
   LIN {X -4.280, Y 45.029, Z 94.350}
   LaserStart_Ext()
   LIN {X -4.280, Y 30.862, Z 94.350}
   LaserEnd_Ext()
   LIN {X -4.280, Y -14.587, Z 94.350}
   LaserStart_Ext()
   LIN {X -4.280, Y -21.866, Z 94.350}
   LaserEnd_Ext()
   LIN {X -3.280, Y -23.320, Z 94.350}
   LaserStart_Ext()
   LIN {X -3.280, Y -11.168, Z 94.350}
   LaserEnd_Ext()
   LIN {X -3.280, Y 27.385, Z 94.350}
   LaserStart_Ext()
   LIN {X -3.280, Y 44.061, Z 94.350}
   LaserEnd_Ext()
   LIN {X -2.280, Y 42.293, Z 94.350}
   LaserStart_Ext()
   LIN {X -2.280, Y 22.393, Z 94.350}
   LaserEnd_Ext()
   LIN {X -2.280, Y -6.977, Z 94.350}
   LaserStart_Ext()
   LIN {X -2.280, Y -15.352, Z 94.350}
   LaserEnd_Ext()
   LIN {X -2.280, Y -21.370, Z 94.350}
   LaserStart_Ext()
   LIN {X -2.280, Y -24.300, Z 94.350}
   LaserEnd_Ext()
   LIN {X -1.280, Y -24.967, Z 94.350}
   LaserStart_Ext()
   LIN {X -1.280, Y -22.532, Z 94.350}
   LaserEnd_Ext()
   LIN {X -1.280, Y -14.209, Z 94.350}
   LaserStart_Ext()
   LIN {X -1.280, Y -1.199, Z 94.350}
   LaserEnd_Ext()
   LIN {X -1.280, Y 16.395, Z 94.350}
   LaserStart_Ext()
   LIN {X -1.280, Y 40.411, Z 94.350}
   LaserEnd_Ext()
   LIN {X -0.280, Y 38.468, Z 94.350}
   LaserStart_Ext()
   LIN {X -0.280, Y -13.311, Z 94.350}
   LaserEnd_Ext()
   LIN {X -0.280, Y -23.370, Z 94.350}
   LaserStart_Ext()
   LIN {X -0.280, Y -25.634, Z 94.350}
   LaserEnd_Ext()
   LIN {X 0.720, Y -25.784, Z 94.350}
   LaserStart_Ext()
   LIN {X 0.720, Y -23.843, Z 94.350}
   LaserEnd_Ext()
   LIN {X 0.720, Y -12.870, Z 94.350}
   LaserStart_Ext()
   LIN {X 0.720, Y 36.308, Z 94.350}
   LaserEnd_Ext()
   LIN {X 1.720, Y 34.135, Z 94.350}
   LaserStart_Ext()
   LIN {X 1.720, Y -12.456, Z 94.350}
   LaserEnd_Ext()
   LIN {X 1.720, Y -24.215, Z 94.350}
   LaserStart_Ext()
   LIN {X 1.720, Y -25.827, Z 94.350}
   LaserEnd_Ext()
   LIN {X 2.720, Y -25.871, Z 94.350}
   LaserStart_Ext()
   LIN {X 2.720, Y -24.235, Z 94.350}
   LaserEnd_Ext()
   LIN {X 2.720, Y -12.444, Z 94.350}
   LaserStart_Ext()
   LIN {X 2.720, Y 31.912, Z 94.350}
   LaserEnd_Ext()
   LIN {X 3.720, Y 29.263, Z 94.350}
   LaserStart_Ext()
   LIN {X 3.720, Y -12.452, Z 94.350}
   LaserEnd_Ext()
   LIN {X 3.720, Y -24.254, Z 94.350}
   LaserStart_Ext()
   LIN {X 3.720, Y -25.913, Z 94.350}
   LaserEnd_Ext()
   LIN {X 4.720, Y -25.931, Z 94.350}
   LaserStart_Ext()
   LIN {X 4.720, Y -23.953, Z 94.350}
   LaserEnd_Ext()
   LIN {X 4.720, Y -12.651, Z 94.350}
   LaserStart_Ext()
   LIN {X 4.720, Y 26.394, Z 94.350}
   LaserEnd_Ext()
   LIN {X 5.720, Y 23.664, Z 94.350}
   LaserStart_Ext()
   LIN {X 5.720, Y -13.129, Z 94.350}
   LaserEnd_Ext()
   LIN {X 5.720, Y -23.530, Z 94.350}
   LaserStart_Ext()
   LIN {X 5.720, Y -25.687, Z 94.350}
   LaserEnd_Ext()
   LIN {X 6.720, Y -25.134, Z 94.350}
   LaserStart_Ext()
   LIN {X 6.720, Y -22.869, Z 94.350}
   LaserEnd_Ext()
   LIN {X 6.720, Y -13.681, Z 94.350}
   LaserStart_Ext()
   LIN {X 6.720, Y 20.655, Z 94.350}
   LaserEnd_Ext()
   LIN {X 7.720, Y 16.703, Z 94.350}
   LaserStart_Ext()
   LIN {X 7.720, Y -14.982, Z 94.350}
   LaserEnd_Ext()
   LIN {X 7.720, Y -21.709, Z 94.350}
   LaserStart_Ext()
   LIN {X 7.720, Y -24.585, Z 94.350}
   LaserEnd_Ext()
   LIN {X 8.720, Y -23.535, Z 94.350}
   LaserStart_Ext()
   LIN {X 8.720, Y -19.407, Z 94.350}
   LaserEnd_Ext()
   LIN {X 8.720, Y -17.353, Z 94.350}
   LaserStart_Ext()
   LIN {X 8.720, Y 12.771, Z 94.350}
